Yaskawa INFORM job: A_ROOF_SIDE_0617_2_PAINT_61.JBI

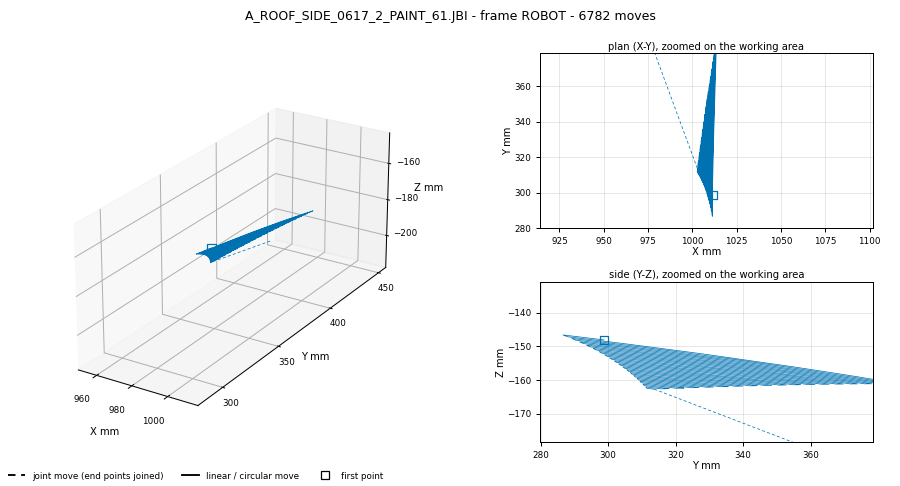
[picture p0: tool path of A_ROOF_SIDE_0617_2_PAINT_61.JBI in frame ROBOT, 6782 of 6782 moves have a stored position in this frame; points joined in program order, loops and branches not executed]
/JOB
//NAME A_ROOF_SIDE_0617_2_PAINT61
//POS
///NPOS 6782,0,0,0,0,0
///TOOL 1
///USER 0
///POSTYPE ROBOT
///RECTAN
///RCONF 1,0,0,0,0,0,0,0,0,0,0,0,0,0,0,0,0,0,0,0,0,0,0,0
C00000=1011.484,298.812,-148.095,169.236,53.491,160.314
C00001=1011.478,298.564,-148.065,169.230,53.497,160.314
C00002=1011.473,298.316,-148.034,169.223,53.504,160.314
C00003=1011.467,298.068,-148.004,169.218,53.510,160.315
C00004=1011.462,297.820,-147.973,169.211,53.517,160.315
C00005=1011.456,297.573,-147.942,169.204,53.524,160.315
C00006=1011.451,297.324,-147.911,169.198,53.530,160.315
C00007=1011.445,297.077,-147.881,169.192,53.537,160.315
C00008=1011.440,296.828,-147.850,169.186,53.544,160.316
C00009=1011.434,296.581,-147.820,169.180,53.551,160.316
C00010=1011.429,296.332,-147.789,169.174,53.558,160.316
C00011=1011.424,296.084,-147.759,169.167,53.565,160.316
C00012=1011.418,295.836,-147.728,169.161,53.572,160.317
C00013=1011.413,295.588,-147.698,169.155,53.578,160.317
C00014=1011.408,295.340,-147.667,169.148,53.585,160.317
C00015=1011.402,295.093,-147.637,169.142,53.592,160.317
C00016=1011.398,294.844,-147.607,169.136,53.599,160.317
C00017=1011.392,294.596,-147.576,169.130,53.605,160.318
C00018=1011.387,294.348,-147.545,169.123,53.612,160.318
C00019=1011.381,294.100,-147.515,169.117,53.620,160.318
C00020=1011.376,293.852,-147.485,169.111,53.626,160.319
C00021=1011.369,293.566,-147.450,169.104,53.634,160.319
C00022=1011.364,293.280,-147.415,169.097,53.642,160.319
C00023=1011.358,292.995,-147.380,169.090,53.650,160.319
C00024=1011.352,292.709,-147.345,169.082,53.658,160.320
C00025=1011.347,292.461,-147.315,169.077,53.665,160.320
C00026=1011.341,292.212,-147.285,169.070,53.672,160.320
C00027=1011.336,291.964,-147.255,169.065,53.679,160.321
C00028=1011.331,291.716,-147.225,169.058,53.686,160.321
C00029=1011.326,291.468,-147.194,169.051,53.693,160.321
C00030=1011.320,291.220,-147.165,169.046,53.700,160.321
C00031=1011.315,290.971,-147.135,169.039,53.707,160.322
C00032=1011.309,290.724,-147.105,169.034,53.714,160.322
C00033=1011.304,290.476,-147.075,169.027,53.721,160.322
C00034=1011.298,290.227,-147.046,169.021,53.728,160.322
C00035=1011.293,289.979,-147.015,169.015,53.736,160.323
C00036=1011.288,289.732,-146.986,169.009,53.742,160.323
C00037=1011.283,289.483,-146.956,169.002,53.750,160.324
C00038=1011.277,289.235,-146.926,168.997,53.757,160.324
C00039=1011.272,288.987,-146.897,168.990,53.764,160.324
C00040=1011.267,288.739,-146.867,168.985,53.771,160.324
C00041=1011.261,288.491,-146.837,168.979,53.779,160.325
C00042=1011.256,288.243,-146.808,168.972,53.785,160.325
C00043=1011.251,287.995,-146.778,168.967,53.793,160.325
C00044=1011.245,287.746,-146.749,168.960,53.800,160.326
C00045=1011.240,287.463,-146.715,168.953,53.808,160.326
C00046=1011.233,287.181,-146.682,168.946,53.816,160.326
C00047=1011.227,286.898,-146.648,168.940,53.824,160.327
C00048=1011.221,286.616,-146.614,168.933,53.833,160.327
C00049=1010.990,287.953,-147.138,168.938,53.865,160.336
C00050=1010.994,288.177,-147.165,168.944,53.858,160.335
C00051=1010.999,288.403,-147.191,168.949,53.852,160.335
C00052=1011.004,288.627,-147.218,168.955,53.845,160.335
C00053=1011.008,288.853,-147.245,168.961,53.839,160.335
C00054=1011.014,289.077,-147.272,168.965,53.832,160.334
C00055=1011.018,289.303,-147.299,168.971,53.826,160.334
C00056=1011.023,289.527,-147.326,168.977,53.819,160.334
C00057=1011.027,289.753,-147.353,168.983,53.813,160.334
C00058=1011.033,290.001,-147.382,168.989,53.806,160.333
C00059=1011.038,290.249,-147.412,168.995,53.799,160.333
C00060=1011.043,290.497,-147.442,169.001,53.792,160.333
C00061=1011.049,290.745,-147.471,169.007,53.785,160.332
C00062=1011.054,290.993,-147.501,169.013,53.778,160.332
C00063=1011.060,291.242,-147.531,169.020,53.770,160.332
C00064=1011.064,291.489,-147.561,169.025,53.764,160.332
C00065=1011.070,291.738,-147.591,169.032,53.756,160.331
C00066=1011.075,291.986,-147.621,169.038,53.749,160.331
C00067=1011.081,292.233,-147.651,169.044,53.743,160.331
C00068=1011.085,292.482,-147.681,169.051,53.736,160.331
C00069=1011.091,292.730,-147.711,169.056,53.728,160.330
C00070=1011.096,293.018,-147.746,169.063,53.720,160.330
C00071=1011.103,293.306,-147.781,169.070,53.712,160.330
C00072=1011.110,293.594,-147.817,169.078,53.704,160.329
C00073=1011.115,293.882,-147.852,169.085,53.696,160.329
C00074=1011.121,294.130,-147.882,169.092,53.689,160.329
C00075=1011.126,294.379,-147.913,169.097,53.683,160.329
C00076=1011.131,294.627,-147.943,169.104,53.676,160.328
C00077=1011.136,294.874,-147.973,169.111,53.669,160.328
C00078=1011.141,295.122,-148.003,169.117,53.662,160.328
C00079=1011.147,295.371,-148.034,169.123,53.655,160.328
C00080=1011.152,295.618,-148.064,169.128,53.648,160.327
C00081=1011.157,295.867,-148.095,169.135,53.641,160.327
C00082=1011.163,296.115,-148.125,169.141,53.635,160.327
C00083=1011.168,296.363,-148.156,169.148,53.628,160.327
C00084=1011.174,296.611,-148.186,169.154,53.621,160.327
C00085=1011.179,296.859,-148.217,169.160,53.614,160.326
C00086=1011.185,297.107,-148.248,169.167,53.607,160.326
C00087=1011.189,297.354,-148.278,169.172,53.601,160.326
C00088=1011.195,297.603,-148.308,169.179,53.594,160.326
C00089=1011.200,297.851,-148.339,169.186,53.587,160.326
C00090=1011.205,298.099,-148.370,169.192,53.581,160.325
C00091=1011.211,298.347,-148.400,169.198,53.574,160.325
C00092=1011.216,298.595,-148.431,169.204,53.567,160.325
C00093=1011.222,298.843,-148.461,169.211,53.560,160.325
C00094=1011.227,299.091,-148.492,169.218,53.554,160.325
C00095=1011.233,299.339,-148.523,169.224,53.547,160.324
C00096=1011.238,299.588,-148.554,169.230,53.540,160.324
C00097=1011.244,299.835,-148.584,169.237,53.534,160.324
C00098=1011.249,300.084,-148.615,169.243,53.527,160.324
C00099=1011.255,300.331,-148.646,169.250,53.520,160.324
C00100=1011.260,300.580,-148.676,169.255,53.514,160.323
C00101=1011.266,300.827,-148.707,169.262,53.507,160.323
C00102=1011.271,301.075,-148.738,169.269,53.500,160.323
C00103=1011.277,301.323,-148.769,169.275,53.494,160.323
C00104=1011.282,301.571,-148.800,169.282,53.487,160.323
C00105=1011.288,301.819,-148.831,169.287,53.480,160.323
C00106=1011.294,302.067,-148.861,169.295,53.474,160.323
C00107=1011.299,302.315,-148.892,169.301,53.467,160.322
C00108=1011.304,302.563,-148.923,169.307,53.461,160.322
C00109=1011.311,302.811,-148.954,169.314,53.454,160.322
C00110=1011.316,303.059,-148.985,169.321,53.448,160.322
C00111=1011.322,303.307,-149.015,169.327,53.441,160.322
C00112=1011.327,303.555,-149.046,169.333,53.434,160.322
C00113=1011.333,303.803,-149.077,169.340,53.428,160.322
C00114=1011.338,304.051,-149.108,169.346,53.422,160.321
C00115=1011.345,304.299,-149.139,169.353,53.415,160.321
C00116=1011.350,304.547,-149.171,169.359,53.409,160.321
C00117=1011.356,304.795,-149.201,169.366,53.402,160.321
C00118=1011.362,305.043,-149.233,169.373,53.395,160.321
C00119=1011.368,305.291,-149.264,169.379,53.389,160.321
C00120=1011.373,305.539,-149.294,169.386,53.382,160.321
C00121=1011.380,305.787,-149.326,169.393,53.376,160.321
C00122=1011.385,306.035,-149.357,169.398,53.370,160.320
C00123=1011.391,306.282,-149.388,169.405,53.363,160.320
C00124=1011.396,306.531,-149.419,169.412,53.356,160.320
C00125=1011.403,306.778,-149.450,169.418,53.350,160.320
C00126=1011.408,307.026,-149.481,169.425,53.344,160.320
C00127=1011.414,307.274,-149.513,169.432,53.337,160.320
C00128=1011.419,307.522,-149.544,169.438,53.331,160.320
C00129=1011.425,307.770,-149.576,169.445,53.325,160.320
C00130=1011.433,308.076,-149.614,169.454,53.316,160.320
C00131=1011.440,308.383,-149.652,169.461,53.309,160.320
C00132=1011.448,308.689,-149.691,169.470,53.301,160.319
C00133=1011.455,308.995,-149.730,169.479,53.293,160.319
C00134=1011.460,309.243,-149.762,169.484,53.287,160.319
C00135=1011.465,309.491,-149.794,169.491,53.281,160.319
C00136=1011.471,309.739,-149.826,169.498,53.275,160.319
C00137=1011.476,309.986,-149.858,169.505,53.269,160.319
C00138=1011.482,310.235,-149.890,169.511,53.263,160.319
C00139=1011.488,310.481,-149.922,169.518,53.256,160.319
C00140=1011.494,310.730,-149.954,169.525,53.250,160.319
C00141=1011.498,310.977,-149.986,169.531,53.244,160.319
C00142=1011.504,311.226,-150.019,169.538,53.238,160.319
C00143=1011.510,311.473,-150.050,169.545,53.232,160.319
C00144=1011.516,311.721,-150.082,169.551,53.225,160.319
C00145=1011.521,311.969,-150.114,169.559,53.219,160.319
C00146=1011.528,312.216,-150.147,169.565,53.213,160.319
C00147=1011.533,312.464,-150.178,169.572,53.207,160.319
C00148=1011.538,312.713,-150.211,169.578,53.201,160.319
C00149=1011.544,312.961,-150.243,169.585,53.195,160.319
C00150=1011.550,313.208,-150.275,169.592,53.189,160.319
C00151=1011.556,313.456,-150.307,169.599,53.183,160.319
C00152=1011.561,313.703,-150.339,169.606,53.177,160.319
C00153=1011.567,313.951,-150.372,169.612,53.171,160.319
C00154=1011.573,314.199,-150.404,169.619,53.165,160.319
C00155=1011.578,314.447,-150.436,169.627,53.158,160.319
C00156=1011.584,314.695,-150.469,169.633,53.153,160.319
C00157=1011.590,314.943,-150.501,169.640,53.146,160.319
C00158=1011.597,315.190,-150.534,169.646,53.141,160.319
C00159=1011.601,315.438,-150.566,169.653,53.134,160.319
C00160=1011.608,315.686,-150.599,169.661,53.128,160.319
C00161=1011.614,315.934,-150.631,169.667,53.123,160.319
C00162=1011.620,316.182,-150.663,169.674,53.116,160.319
C00163=1011.625,316.429,-150.695,169.681,53.110,160.319
C00164=1011.632,316.677,-150.728,169.688,53.105,160.319
C00165=1011.637,316.925,-150.760,169.695,53.099,160.319
C00166=1011.643,317.173,-150.793,169.701,53.093,160.319
C00167=1011.649,317.421,-150.825,169.709,53.087,160.319
C00168=1011.655,317.668,-150.857,169.716,53.081,160.319
C00169=1011.661,317.916,-150.890,169.722,53.076,160.319
C00170=1011.667,318.164,-150.922,169.730,53.069,160.319
C00171=1011.673,318.412,-150.956,169.737,53.063,160.319
C00172=1011.679,318.659,-150.988,169.743,53.057,160.319
C00173=1011.685,318.907,-151.020,169.751,53.052,160.319
C00174=1011.691,319.155,-151.053,169.758,53.046,160.320
C00175=1011.698,319.403,-151.086,169.764,53.040,160.319
C00176=1011.703,319.651,-151.118,169.771,53.034,160.319
C00177=1011.709,319.899,-151.151,169.779,53.028,160.320
C00178=1011.715,320.146,-151.184,169.785,53.023,160.320
C00179=1011.722,320.394,-151.217,169.792,53.016,160.320
C00180=1011.728,320.642,-151.249,169.800,53.011,160.320
C00181=1011.734,320.889,-151.282,169.806,53.005,160.320
C00182=1011.739,321.138,-151.315,169.814,53.000,160.320
C00183=1011.746,321.385,-151.348,169.821,52.994,160.320
C00184=1011.752,321.633,-151.380,169.827,52.988,160.320
C00185=1011.758,321.880,-151.413,169.835,52.982,160.320
C00186=1011.765,322.128,-151.446,169.842,52.976,160.320
C00187=1011.770,322.376,-151.479,169.849,52.971,160.321
C00188=1011.777,322.624,-151.512,169.856,52.965,160.321
C00189=1011.783,322.871,-151.545,169.864,52.959,160.321
C00190=1011.791,323.183,-151.586,169.873,52.952,160.321
C00191=1011.799,323.495,-151.627,169.882,52.945,160.321
C00192=1011.807,323.807,-151.669,169.891,52.938,160.321
C00193=1011.815,324.119,-151.711,169.900,52.931,160.322
C00194=1011.821,324.366,-151.743,169.906,52.925,160.321
C00195=1011.827,324.614,-151.776,169.914,52.920,160.322
C00196=1011.833,324.862,-151.810,169.921,52.914,160.322
C00197=1011.839,325.109,-151.842,169.929,52.908,160.322
C00198=1011.847,325.357,-151.876,169.936,52.903,160.322
C00199=1011.853,325.604,-151.909,169.943,52.897,160.322
C00200=1011.859,325.852,-151.943,169.951,52.891,160.322
C00201=1011.864,326.100,-151.976,169.957,52.886,160.323
C00202=1011.871,326.347,-152.010,169.965,52.881,160.323
C00203=1011.877,326.595,-152.043,169.973,52.875,160.323
C00204=1011.883,326.843,-152.077,169.979,52.870,160.323
C00205=1011.889,327.090,-152.110,169.986,52.864,160.323
C00206=1011.896,327.338,-152.145,169.994,52.859,160.324
C00207=1011.901,327.586,-152.178,170.001,52.854,160.324
C00208=1011.908,327.833,-152.211,170.008,52.848,160.324
C00209=1011.914,328.081,-152.246,170.016,52.843,160.324
C00210=1011.920,328.329,-152.279,170.023,52.838,160.324
C00211=1011.926,328.576,-152.313,170.030,52.832,160.325
C00212=1011.933,328.824,-152.347,170.038,52.827,160.325
C00213=1011.939,329.071,-152.380,170.046,52.821,160.325
C00214=1011.946,329.319,-152.414,170.052,52.816,160.325
C00215=1011.951,329.567,-152.448,170.060,52.811,160.325
C00216=1011.958,329.814,-152.481,170.068,52.805,160.326
C00217=1011.964,330.062,-152.515,170.074,52.800,160.326
C00218=1011.970,330.310,-152.550,170.082,52.795,160.326
C00219=1011.977,330.557,-152.583,170.090,52.789,160.326
C00220=1011.983,330.804,-152.617,170.097,52.784,160.327
C00221=1011.990,331.052,-152.652,170.104,52.778,160.327
C00222=1011.996,331.299,-152.685,170.112,52.773,160.327
C00223=1012.002,331.548,-152.719,170.119,52.768,160.327
C00224=1012.008,331.795,-152.753,170.127,52.762,160.327
C00225=1012.016,332.042,-152.788,170.134,52.757,160.328
C00226=1012.022,332.290,-152.822,170.142,52.752,160.328
C00227=1012.028,332.538,-152.856,170.150,52.747,160.328
C00228=1012.034,332.786,-152.890,170.156,52.742,160.328
C00229=1012.040,333.033,-152.924,170.164,52.736,160.329
C00230=1012.047,333.281,-152.959,170.172,52.731,160.329
C00231=1012.053,333.528,-152.993,170.180,52.726,160.329
C00232=1012.059,333.776,-153.028,170.186,52.721,160.330
C00233=1012.066,334.024,-153.063,170.194,52.716,160.330
C00234=1012.072,334.271,-153.097,170.202,52.711,160.330
C00235=1012.079,334.519,-153.130,170.210,52.705,160.330
C00236=1012.086,334.766,-153.166,170.217,52.701,160.331
C00237=1012.092,335.013,-153.200,170.225,52.695,160.331
C00238=1012.098,335.261,-153.234,170.233,52.691,160.332
C00239=1012.105,335.509,-153.269,170.240,52.685,160.332
C00240=1012.111,335.756,-153.303,170.248,52.681,160.332
C00241=1012.117,336.003,-153.338,170.255,52.675,160.332
C00242=1012.124,336.251,-153.373,170.263,52.670,160.333
C00243=1012.130,336.499,-153.407,170.271,52.665,160.333
C00244=1012.137,336.746,-153.442,170.278,52.661,160.333
C00245=1012.144,336.993,-153.476,170.286,52.655,160.334
C00246=1012.150,337.241,-153.511,170.294,52.650,160.334
C00247=1012.157,337.489,-153.545,170.302,52.645,160.334
C00248=1012.164,337.736,-153.580,170.310,52.640,160.335
C00249=1012.170,337.984,-153.616,170.316,52.635,160.335
C00250=1012.178,338.291,-153.658,170.326,52.629,160.335
C00251=1012.186,338.599,-153.702,170.336,52.623,160.336
C00252=1012.194,338.907,-153.745,170.346,52.617,160.337
C00253=1012.202,339.213,-153.789,170.355,52.611,160.337
C00254=1012.209,339.461,-153.824,170.364,52.606,160.337
C00255=1012.216,339.708,-153.859,170.371,52.601,160.338
C00256=1012.223,339.956,-153.894,170.378,52.596,160.338
C00257=1012.229,340.203,-153.930,170.386,52.591,160.338
C00258=1012.235,340.451,-153.965,170.395,52.587,160.339
C00259=1012.242,340.699,-154.000,170.403,52.582,160.339
C00260=1012.249,340.946,-154.035,170.410,52.576,160.340
C00261=1012.255,341.193,-154.070,170.418,52.572,160.340
C00262=1012.262,341.441,-154.105,170.426,52.567,160.340
C00263=1012.268,341.688,-154.141,170.434,52.562,160.341
C00264=1012.275,341.935,-154.177,170.442,52.558,160.341
C00265=1012.282,342.182,-154.212,170.450,52.553,160.342
C00266=1012.289,342.430,-154.247,170.458,52.548,160.342
C00267=1012.296,342.677,-154.282,170.465,52.544,160.343
C00268=1012.302,342.925,-154.318,170.473,52.539,160.343
C00269=1012.309,343.173,-154.353,170.481,52.534,160.344
C00270=1012.316,343.420,-154.389,170.490,52.529,160.344
C00271=1012.323,343.667,-154.424,170.498,52.525,160.344
C00272=1012.329,343.915,-154.460,170.506,52.520,160.345
C00273=1012.336,344.162,-154.495,170.514,52.515,160.345
C00274=1012.343,344.409,-154.531,170.521,52.511,160.346
C00275=1012.350,344.657,-154.566,170.530,52.506,160.346
C00276=1012.356,344.905,-154.602,170.538,52.502,160.347
C00277=1012.363,345.151,-154.638,170.546,52.497,160.347
C00278=1012.370,345.399,-154.673,170.554,52.492,160.348
C00279=1012.378,345.646,-154.709,170.562,52.487,160.348
C00280=1012.384,345.894,-154.745,170.571,52.483,160.349
C00281=1012.391,346.141,-154.781,170.579,52.478,160.349
C00282=1012.397,346.388,-154.816,170.587,52.474,160.350
C00283=1012.404,346.636,-154.853,170.594,52.469,160.350
C00284=1012.411,346.883,-154.888,170.602,52.465,160.351
C00285=1012.417,347.130,-154.924,170.611,52.460,160.351
C00286=1012.425,347.378,-154.961,170.619,52.456,160.352
C00287=1012.431,347.625,-154.996,170.627,52.451,160.352
C00288=1012.438,347.872,-155.032,170.635,52.447,160.353
C00289=1012.445,348.120,-155.069,170.644,52.443,160.353
C00290=1012.452,348.366,-155.105,170.652,52.438,160.354
C00291=1012.459,348.614,-155.142,170.661,52.434,160.355
C00292=1012.466,348.862,-155.177,170.669,52.429,160.355
C00293=1012.472,349.109,-155.213,170.676,52.425,160.356
C00294=1012.480,349.356,-155.250,170.684,52.420,160.356
C00295=1012.486,349.603,-155.286,170.693,52.416,160.357
C00296=1012.494,349.851,-155.322,170.701,52.412,160.357
C00297=1012.500,350.098,-155.359,170.710,52.407,160.358
C00298=1012.508,350.345,-155.395,170.718,52.403,160.358
C00299=1012.514,350.592,-155.431,170.726,52.399,160.359
C00300=1012.522,350.840,-155.468,170.735,52.394,160.360
C00301=1012.528,351.087,-155.504,170.743,52.390,160.360
C00302=1012.536,351.334,-155.540,170.751,52.386,160.361
C00303=1012.543,351.582,-155.577,170.760,52.381,160.361
C00304=1012.550,351.828,-155.614,170.768,52.377,160.362
C00305=1012.557,352.076,-155.650,170.777,52.373,160.362
C00306=1012.564,352.322,-155.686,170.785,52.368,160.363
C00307=1012.571,352.570,-155.723,170.794,52.364,160.364
C00308=1012.579,352.818,-155.759,170.802,52.360,160.364
C00309=1012.586,353.064,-155.796,170.810,52.355,160.365
C00310=1012.594,353.369,-155.842,170.821,52.351,160.366
C00311=1012.603,353.675,-155.887,170.832,52.346,160.367
C00312=1012.612,353.979,-155.932,170.842,52.340,160.367
C00313=1012.621,354.284,-155.978,170.852,52.335,160.368
C00314=1012.628,354.531,-156.015,170.861,52.331,160.369
C00315=1012.634,354.778,-156.052,170.869,52.327,160.369
C00316=1012.642,355.025,-156.089,170.879,52.322,160.370
C00317=1012.649,355.273,-156.125,170.887,52.318,160.371
C00318=1012.657,355.520,-156.163,170.896,52.314,160.371
C00319=1012.665,355.767,-156.200,170.904,52.310,160.372
C00320=1012.671,356.014,-156.236,170.913,52.306,160.373
C00321=1012.678,356.261,-156.274,170.922,52.302,160.373
C00322=1012.685,356.508,-156.311,170.930,52.298,160.374
C00323=1012.693,356.756,-156.348,170.939,52.294,160.375
C00324=1012.700,357.003,-156.385,170.948,52.290,160.376
C00325=1012.708,357.250,-156.423,170.956,52.286,160.376
C00326=1012.715,357.497,-156.460,170.965,52.282,160.377
C00327=1012.723,357.744,-156.497,170.973,52.278,160.378
C00328=1012.730,357.992,-156.534,170.982,52.274,160.378
C00329=1012.737,358.239,-156.571,170.991,52.270,160.379
C00330=1012.744,358.486,-156.609,171.000,52.266,160.380
C00331=1012.752,358.733,-156.647,171.009,52.262,160.381
C00332=1012.758,358.979,-156.684,171.018,52.258,160.381
C00333=1012.766,359.226,-156.722,171.026,52.254,160.382
C00334=1012.773,359.473,-156.759,171.035,52.251,160.383
C00335=1012.781,359.721,-156.797,171.044,52.247,160.384
C00336=1012.788,359.968,-156.835,171.053,52.243,160.384
C00337=1012.795,360.215,-156.872,171.061,52.239,160.385
C00338=1012.803,360.462,-156.911,171.070,52.235,160.386
C00339=1012.810,360.709,-156.948,171.080,52.231,160.387
C00340=1012.817,360.956,-156.986,171.089,52.227,160.388
C00341=1012.825,361.203,-157.024,171.098,52.224,160.389
C00342=1012.832,361.450,-157.061,171.106,52.220,160.389
C00343=1012.839,361.697,-157.099,171.115,52.216,160.390
C00344=1012.847,361.943,-157.137,171.124,52.212,160.391
C00345=1012.855,362.191,-157.175,171.134,52.208,160.392
C00346=1012.862,362.438,-157.213,171.143,52.205,160.393
C00347=1012.870,362.685,-157.251,171.151,52.201,160.393
C00348=1012.877,362.931,-157.289,171.160,52.197,160.394
C00349=1012.885,363.179,-157.327,171.169,52.194,160.395
C00350=1012.892,363.426,-157.365,171.179,52.190,160.396
C00351=1012.900,363.673,-157.403,171.188,52.186,160.397
C00352=1012.907,363.919,-157.441,171.197,52.183,160.397
C00353=1012.915,364.167,-157.480,171.206,52.179,160.398
C00354=1012.923,364.414,-157.517,171.216,52.175,160.399
C00355=1012.930,364.660,-157.555,171.225,52.172,160.400
C00356=1012.938,364.907,-157.594,171.234,52.168,160.401
C00357=1012.946,365.155,-157.632,171.243,52.165,160.402
C00358=1012.954,365.402,-157.670,171.253,52.161,160.403
C00359=1012.961,365.648,-157.708,171.262,52.157,160.404
C00360=1012.969,365.895,-157.747,171.271,52.154,160.405
C00361=1012.977,366.142,-157.785,171.280,52.151,160.405
C00362=1012.985,366.389,-157.824,171.290,52.147,160.406
C00363=1012.993,366.636,-157.862,171.299,52.143,160.407
C00364=1013.000,366.883,-157.901,171.308,52.140,160.408
C00365=1013.008,367.130,-157.940,171.318,52.136,160.409
C00366=1013.015,367.376,-157.978,171.327,52.132,160.410
C00367=1013.023,367.624,-158.017,171.336,52.129,160.411
C00368=1013.030,367.870,-158.055,171.346,52.126,160.412
C00369=1013.039,368.117,-158.095,171.355,52.122,160.413
C00370=1013.048,368.429,-158.144,171.367,52.118,160.414
C00371=1013.057,368.742,-158.193,171.379,52.114,160.415
C00372=1013.067,369.055,-158.242,171.390,52.109,160.416
C00373=1013.077,369.367,-158.291,171.403,52.105,160.418
C00374=1013.085,369.614,-158.331,171.413,52.102,160.419
C00375=1013.093,369.860,-158.369,171.422,52.098,160.420
C00376=1013.101,370.107,-158.409,171.431,52.095,160.421
C00377=1013.108,370.355,-158.448,171.441,52.091,160.422
C00378=1013.117,370.601,-158.487,171.450,52.089,160.423
C00379=1013.124,370.848,-158.525,171.460,52.085,160.424
C00380=1013.132,371.095,-158.565,171.470,52.082,160.425
C00381=1013.140,371.342,-158.604,171.479,52.078,160.426
C00382=1013.149,371.588,-158.643,171.489,52.075,160.427
C00383=1013.156,371.835,-158.683,171.498,52.072,160.428
C00384=1013.164,372.082,-158.721,171.508,52.068,160.429
C00385=1013.172,372.329,-158.761,171.518,52.066,160.430
C00386=1013.180,372.575,-158.801,171.528,52.062,160.431
C00387=1013.189,372.822,-158.840,171.537,52.059,160.432
C00388=1013.196,373.069,-158.879,171.548,52.056,160.433
C00389=1013.205,373.316,-158.918,171.557,52.053,160.434
C00390=1013.212,373.562,-158.957,171.567,52.049,160.435
C00391=1013.220,373.809,-158.997,171.576,52.046,160.436
C00392=1013.229,374.055,-159.037,171.587,52.043,160.438
C00393=1013.237,374.302,-159.076,171.596,52.040,160.439
C00394=1013.245,374.549,-159.116,171.606,52.037,160.440
C00395=1013.253,374.796,-159.155,171.616,52.034,160.441
C00396=1013.262,375.042,-159.195,171.626,52.031,160.442
C00397=1013.269,375.289,-159.234,171.636,52.028,160.443
C00398=1013.277,375.536,-159.274,171.646,52.025,160.444
C00399=1013.285,375.782,-159.315,171.655,52.022,160.445
C00400=1013.294,376.030,-159.355,171.666,52.019,160.447
C00401=1013.302,376.276,-159.395,171.676,52.015,160.448
C00402=1013.310,376.523,-159.435,171.686,52.013,160.449
C00403=1013.318,376.769,-159.475,171.696,52.009,160.450
C00404=1013.326,377.016,-159.515,171.705,52.007,160.451
C00405=1013.334,377.263,-159.555,171.716,52.004,160.453
C00406=1013.343,377.508,-159.595,171.727,52.001,160.454
C00407=1013.351,377.755,-159.635,171.736,51.998,160.455
C00408=1013.359,378.002,-159.676,171.746,51.995,160.456
C00409=1013.368,378.249,-159.715,171.756,51.992,160.457
C00410=1013.376,378.495,-159.756,171.767,51.989,160.458
C00411=1013.384,378.742,-159.797,171.777,51.986,160.460
C00412=1013.392,378.988,-159.837,171.787,51.984,160.461
C00413=1013.401,379.235,-159.877,171.797,51.980,160.462
C00414=1013.409,379.481,-159.918,171.808,51.978,160.463
C00415=1013.417,379.728,-159.958,171.817,51.975,160.465
C00416=1013.426,379.975,-159.998,171.828,51.972,160.466
C00417=1013.434,380.221,-160.039,171.839,51.969,160.467
C00418=1013.442,380.468,-160.079,171.849,51.967,160.468
C00419=1013.451,380.714,-160.120,171.859,51.964,160.470
C00420=1013.459,380.961,-160.160,171.870,51.961,160.471
C00421=1013.468,381.207,-160.201,171.880,51.958,160.472
C00422=1013.477,381.453,-160.241,171.891,51.955,160.473
C00423=1013.485,381.700,-160.282,171.901,51.953,160.475
C00424=1013.493,381.947,-160.323,171.911,51.950,160.476
C00425=1013.503,382.193,-160.363,171.922,51.947,160.477
C00426=1013.511,382.440,-160.404,171.933,51.945,160.479
C00427=1013.520,382.687,-160.445,171.943,51.942,160.480
C00428=1013.528,382.933,-160.485,171.954,51.939,160.481
C00429=1013.537,383.179,-160.527,171.964,51.936,160.483
C00430=1013.548,383.480,-160.577,171.977,51.934,160.484
C00431=1013.558,383.781,-160.627,171.990,51.930,160.486
C00432=1013.569,384.083,-160.677,172.003,51.927,160.488
C00433=1013.580,384.384,-160.727,172.017,51.924,160.489
C00434=1013.588,384.631,-160.768,172.027,51.921,160.491
C00435=1013.597,384.877,-160.809,172.037,51.919,160.492
C00436=1013.606,385.124,-160.850,172.048,51.916,160.494
C00437=1013.615,385.370,-160.892,172.059,51.914,160.495
C00438=1013.623,385.616,-160.933,172.070,51.911,160.496
C00439=1013.632,385.863,-160.974,172.080,51.908,160.498
C00440=1013.640,386.109,-161.016,172.092,51.906,160.499
C00441=1013.649,386.356,-161.058,172.103,51.904,160.501
C00442=1013.305,384.294,-161.060,171.994,51.982,160.501
C00443=1013.295,384.035,-161.017,171.984,51.985,160.499
C00444=1013.286,383.776,-160.974,171.972,51.988,160.498
C00445=1013.277,383.517,-160.931,171.961,51.991,160.496
C00446=1013.268,383.257,-160.887,171.949,51.994,160.495
C00447=1013.259,383.011,-160.847,171.939,51.996,160.494
C00448=1013.250,382.764,-160.806,171.929,51.999,160.492
C00449=1013.242,382.518,-160.765,171.918,52.001,160.491
C00450=1013.233,382.271,-160.725,171.907,52.005,160.490
C00451=1013.225,382.025,-160.684,171.897,52.007,160.488
C00452=1013.216,381.778,-160.643,171.886,52.010,160.487
C00453=1013.208,381.532,-160.603,171.875,52.013,160.486
C00454=1013.200,381.285,-160.563,171.865,52.015,160.484
C00455=1013.191,381.038,-160.522,171.855,52.018,160.483
C00456=1013.182,380.792,-160.482,171.844,52.021,160.482
C00457=1013.174,380.545,-160.441,171.833,52.024,160.480
C00458=1013.165,380.299,-160.400,171.824,52.027,160.479
C00459=1013.157,380.053,-160.360,171.813,52.029,160.478
C00460=1013.148,379.806,-160.320,171.803,52.032,160.477
C00461=1013.140,379.559,-160.279,171.792,52.035,160.475
C00462=1013.132,379.313,-160.239,171.783,52.038,160.474
C00463=1013.123,379.066,-160.198,171.772,52.041,160.473
C00464=1013.115,378.819,-160.158,171.761,52.044,160.472
C00465=1013.107,378.573,-160.118,171.751,52.047,160.470
C00466=1013.099,378.326,-160.078,171.742,52.050,160.469
C00467=1013.090,378.079,-160.037,171.731,52.052,160.468
C00468=1013.082,377.833,-159.998,171.721,52.056,160.467
C00469=1013.074,377.587,-159.957,171.711,52.059,160.466
C00470=1013.066,377.340,-159.917,171.701,52.062,160.465
C00471=1013.058,377.093,-159.876,171.690,52.064,160.463
C00472=1013.049,376.847,-159.837,171.680,52.067,160.462
C00473=1013.041,376.601,-159.797,171.670,52.071,160.461
C00474=1013.034,376.354,-159.757,171.661,52.073,160.460
C00475=1013.025,376.107,-159.717,171.650,52.077,160.459
C00476=1013.017,375.861,-159.677,171.640,52.080,160.457
C00477=1013.009,375.613,-159.636,171.631,52.083,160.456
C00478=1013.001,375.367,-159.597,171.620,52.086,160.455
C00479=1012.993,375.120,-159.557,171.611,52.089,160.454
C00480=1012.985,374.874,-159.517,171.600,52.092,160.453
C00481=1012.977,374.627,-159.478,171.591,52.095,160.452
C00482=1012.969,374.380,-159.439,171.581,52.098,160.451
C00483=1012.961,374.133,-159.399,171.570,52.101,160.449
C00484=1012.953,373.887,-159.360,171.561,52.104,160.448
C00485=1012.944,373.640,-159.320,171.551,52.108,160.447
C00486=1012.936,373.393,-159.280,171.541,52.111,160.446
C00487=1012.928,373.147,-159.241,171.531,52.114,160.445
C00488=1012.919,372.900,-159.202,171.522,52.117,160.444
C00489=1012.912,372.653,-159.163,171.512,52.121,160.443
C00490=1012.904,372.406,-159.123,171.502,52.124,160.442
C00491=1012.895,372.159,-159.084,171.492,52.128,160.441
C00492=1012.888,371.913,-159.045,171.483,52.130,160.440
C00493=1012.880,371.666,-159.006,171.473,52.134,160.439
C00494=1012.872,371.419,-158.966,171.464,52.137,160.438
C00495=1012.864,371.172,-158.927,171.453,52.140,160.437
C00496=1012.856,370.926,-158.888,171.444,52.144,160.436
C00497=1012.849,370.678,-158.849,171.434,52.147,160.435
C00498=1012.840,370.432,-158.810,171.425,52.151,160.434
C00499=1012.833,370.185,-158.772,171.414,52.154,160.433
C00500=1012.825,369.938,-158.732,171.405,52.157,160.432
C00501=1012.817,369.691,-158.693,171.396,52.160,160.431
C00502=1012.809,369.445,-158.654,171.386,52.164,160.430
C00503=1012.799,369.130,-158.604,171.374,52.169,160.429
C00504=1012.789,368.815,-158.555,171.362,52.173,160.427
C00505=1012.779,368.500,-158.505,171.350,52.177,160.426
C00506=1012.770,368.186,-158.455,171.338,52.182,160.425
C00507=1012.762,367.939,-158.417,171.328,52.185,160.424
C00508=1012.754,367.692,-158.378,171.319,52.188,160.423
C00509=1012.747,367.445,-158.339,171.309,52.192,160.422
C00510=1012.739,367.198,-158.301,171.300,52.196,160.421
C00511=1012.731,366.951,-158.263,171.292,52.199,160.420
C00512=1012.724,366.704,-158.223,171.281,52.202,160.419
C00513=1012.717,366.457,-158.185,171.272,52.206,160.418
C00514=1012.709,366.211,-158.147,171.263,52.209,160.417
C00515=1012.701,365.964,-158.108,171.253,52.213,160.416
C00516=1012.693,365.717,-158.070,171.244,52.217,160.415
C00517=1012.685,365.470,-158.031,171.236,52.221,160.415
C00518=1012.678,365.223,-157.994,171.226,52.225,160.414
C00519=1012.670,364.976,-157.955,171.217,52.228,160.413
C00520=1012.662,364.729,-157.917,171.208,52.232,160.412
C00521=1012.655,364.482,-157.880,171.198,52.235,160.411
C00522=1012.647,364.235,-157.841,171.189,52.239,160.410
C00523=1012.639,363.988,-157.803,171.180,52.242,160.409
C00524=1012.632,363.741,-157.765,171.171,52.246,160.408
C00525=1012.624,363.495,-157.727,171.161,52.250,160.408
C00526=1012.617,363.247,-157.689,171.152,52.254,160.407
C00527=1012.609,363.000,-157.651,171.143,52.257,160.406
C00528=1012.602,362.753,-157.613,171.134,52.261,160.405
C00529=1012.594,362.507,-157.575,171.125,52.265,160.404
C00530=1012.587,362.259,-157.537,171.116,52.269,160.403
C00531=1012.579,362.012,-157.499,171.107,52.272,160.402
C00532=1012.572,361.765,-157.461,171.098,52.276,160.402
C00533=1012.564,361.518,-157.424,171.088,52.280,160.401
C00534=1012.557,361.271,-157.386,171.080,52.284,160.400
C00535=1012.550,361.024,-157.348,171.071,52.288,160.399
C00536=1012.542,360.777,-157.311,171.062,52.292,160.399
C00537=1012.535,360.531,-157.272,171.053,52.295,160.398
C00538=1012.528,360.283,-157.235,171.045,52.300,160.397
C00539=1012.520,360.036,-157.197,171.035,52.303,160.396
C00540=1012.513,359.789,-157.160,171.026,52.308,160.395
C00541=1012.506,359.542,-157.122,171.017,52.311,160.395
C00542=1012.499,359.295,-157.085,171.009,52.315,160.394
C00543=1012.491,359.048,-157.046,171.000,52.319,160.393
C00544=1012.484,358.801,-157.009,170.991,52.323,160.392
C00545=1012.477,358.554,-156.971,170.982,52.327,160.392
C00546=1012.469,358.307,-156.934,170.973,52.331,160.391
C00547=1012.462,358.059,-156.897,170.964,52.335,160.390
C00548=1012.455,357.812,-156.859,170.956,52.339,160.389
C00549=1012.448,357.565,-156.822,170.947,52.343,160.389
C00550=1012.440,357.318,-156.785,170.938,52.347,160.388
C00551=1012.433,357.071,-156.747,170.930,52.351,160.387
C00552=1012.426,356.823,-156.711,170.921,52.355,160.387
C00553=1012.418,356.576,-156.673,170.911,52.359,160.386
C00554=1012.411,356.330,-156.637,170.903,52.363,160.385
C00555=1012.404,356.082,-156.600,170.894,52.368,160.384
C00556=1012.397,355.835,-156.562,170.886,52.372,160.384
C00557=1012.390,355.588,-156.525,170.877,52.376,160.383
C00558=1012.382,355.341,-156.489,170.869,52.380,160.382
C00559=1012.375,355.094,-156.451,170.860,52.384,160.382
C00560=1012.368,354.846,-156.415,170.852,52.388,160.381
C00561=1012.360,354.600,-156.378,170.843,52.392,160.380
C00562=1012.353,354.352,-156.341,170.835,52.396,160.380
C00563=1012.345,354.045,-156.295,170.823,52.402,160.379
C00564=1012.336,353.738,-156.249,170.812,52.407,160.378
C00565=1012.327,353.430,-156.204,170.802,52.412,160.377
C00566=1012.319,353.124,-156.158,170.792,52.417,160.376
C00567=1012.311,352.876,-156.122,170.783,52.421,160.376
C00568=1012.304,352.630,-156.084,170.775,52.425,160.375
C00569=1012.298,352.382,-156.048,170.767,52.430,160.375
C00570=1012.290,352.135,-156.011,170.758,52.434,160.374
C00571=1012.283,351.888,-155.975,170.749,52.438,160.373
C00572=1012.276,351.640,-155.939,170.741,52.443,160.373
C00573=1012.269,351.393,-155.902,170.733,52.447,160.372
C00574=1012.262,351.146,-155.866,170.724,52.451,160.372
C00575=1012.255,350.899,-155.830,170.716,52.456,160.371
C00576=1012.248,350.651,-155.793,170.708,52.460,160.370
C00577=1012.241,350.404,-155.757,170.699,52.464,160.370
C00578=1012.234,350.157,-155.721,170.691,52.469,160.369
C00579=1012.227,349.910,-155.684,170.682,52.473,160.369
C00580=1012.220,349.662,-155.648,170.674,52.478,160.368
C00581=1012.213,349.415,-155.612,170.666,52.482,160.368
C00582=1012.206,349.168,-155.575,170.658,52.487,160.367
C00583=1012.199,348.921,-155.539,170.649,52.491,160.366
C00584=1012.192,348.672,-155.503,170.641,52.496,160.366
C00585=1012.186,348.425,-155.467,170.632,52.500,160.365
C00586=1012.179,348.179,-155.431,170.624,52.505,160.365
C00587=1012.172,347.931,-155.394,170.616,52.509,160.364
C00588=1012.165,347.684,-155.359,170.608,52.514,160.364
C00589=1012.159,347.436,-155.323,170.599,52.518,160.363
C00590=1012.151,347.189,-155.287,170.591,52.523,160.363
C00591=1012.144,346.942,-155.251,170.583,52.527,160.362
C00592=1012.138,346.695,-155.215,170.574,52.532,160.361
C00593=1012.130,346.447,-155.179,170.566,52.536,160.361
C00594=1012.124,346.199,-155.143,170.558,52.541,160.361
C00595=1012.117,345.953,-155.107,170.551,52.546,160.360
C00596=1012.110,345.705,-155.072,170.542,52.550,160.360
C00597=1012.104,345.458,-155.036,170.534,52.554,160.359
C00598=1012.097,345.210,-155.000,170.526,52.559,160.359
C00599=1012.090,344.963,-154.965,170.518,52.564,160.358
C00600=1012.083,344.716,-154.929,170.510,52.569,160.358
C00601=1012.077,344.468,-154.893,170.502,52.574,160.357
C00602=1012.070,344.221,-154.858,170.493,52.578,160.357
C00603=1012.063,343.973,-154.823,170.485,52.583,160.356
C00604=1012.055,343.726,-154.787,170.477,52.587,160.356
C00605=1012.049,343.479,-154.751,170.469,52.592,160.355
C00606=1012.043,343.231,-154.716,170.462,52.597,160.355
C00607=1012.036,342.984,-154.681,170.454,52.601,160.354
C00608=1012.029,342.737,-154.646,170.446,52.606,160.354
C00609=1012.023,342.489,-154.610,170.438,52.611,160.353
C00610=1012.016,342.242,-154.574,170.429,52.616,160.353
C00611=1012.009,341.995,-154.539,170.421,52.620,160.353
C00612=1012.003,341.747,-154.504,170.413,52.625,160.352
C00613=1011.996,341.500,-154.469,170.407,52.630,160.352
C00614=1011.990,341.252,-154.433,170.398,52.635,160.352
C00615=1011.983,341.005,-154.398,170.390,52.640,160.351
C00616=1011.976,340.758,-154.363,170.382,52.645,160.351
C00617=1011.970,340.510,-154.328,170.374,52.650,160.350
C00618=1011.963,340.262,-154.293,170.366,52.654,160.350
C00619=1011.956,340.015,-154.258,170.358,52.660,160.349
C00620=1011.950,339.767,-154.222,170.351,52.664,160.349
C00621=1011.943,339.520,-154.187,170.343,52.669,160.349
C00622=1011.937,339.272,-154.152,170.335,52.674,160.348
C00623=1011.929,338.963,-154.109,170.325,52.680,160.348
C00624=1011.920,338.653,-154.064,170.316,52.686,160.347
C00625=1011.912,338.343,-154.021,170.306,52.692,160.347
C00626=1011.904,338.033,-153.978,170.296,52.699,160.346
C00627=1011.898,337.786,-153.943,170.288,52.703,160.346
C00628=1011.891,337.538,-153.908,170.280,52.709,160.346
C00629=1011.884,337.291,-153.873,170.272,52.714,160.345
C00630=1011.878,337.043,-153.839,170.266,52.719,160.345
C00631=1011.872,336.796,-153.804,170.258,52.724,160.345
C00632=1011.865,336.548,-153.770,170.250,52.729,160.344
C00633=1011.859,336.301,-153.735,170.242,52.734,160.344
C00634=1011.851,336.053,-153.701,170.234,52.739,160.344
C00635=1011.846,335.806,-153.667,170.226,52.744,160.343
C00636=1011.839,335.558,-153.631,170.219,52.749,160.343
C00637=1011.832,335.310,-153.597,170.211,52.754,160.343
C00638=1011.826,335.063,-153.563,170.204,52.760,160.342
C00639=1011.820,334.816,-153.528,170.195,52.764,160.342
C00640=1011.813,334.568,-153.493,170.189,52.769,160.342
C00641=1011.807,334.321,-153.459,170.181,52.775,160.342
C00642=1011.801,334.073,-153.425,170.173,52.780,160.341
C00643=1011.794,333.825,-153.390,170.165,52.785,160.341
C00644=1011.787,333.578,-153.356,170.158,52.791,160.341
C00645=1011.781,333.330,-153.322,170.151,52.795,160.340
C00646=1011.775,333.083,-153.288,170.143,52.801,160.340
C00647=1011.769,332.835,-153.254,170.135,52.806,160.340
C00648=1011.763,332.588,-153.219,170.128,52.811,160.339
C00649=1011.756,332.340,-153.185,170.120,52.816,160.339
C00650=1011.751,332.092,-153.151,170.113,52.821,160.339
C00651=1011.744,331.844,-153.117,170.105,52.827,160.339
C00652=1011.738,331.597,-153.083,170.097,52.832,160.338
C00653=1011.731,331.349,-153.049,170.091,52.837,160.338
C00654=1011.725,331.102,-153.015,170.083,52.843,160.338
C00655=1011.718,330.855,-152.981,170.075,52.848,160.337
C00656=1011.712,330.607,-152.947,170.067,52.853,160.337
C00657=1011.706,330.359,-152.912,170.061,52.858,160.337
C00658=1011.699,330.112,-152.880,170.053,52.864,160.337
C00659=1011.693,329.864,-152.845,170.045,52.869,160.337
C00660=1011.687,329.616,-152.811,170.038,52.875,160.336
C00661=1011.680,329.369,-152.778,170.031,52.880,160.336
C00662=1011.674,329.121,-152.744,170.023,52.885,160.336
C00663=1011.668,328.874,-152.710,170.016,52.891,160.336
C00664=1011.661,328.626,-152.676,170.008,52.896,160.335
C00665=1011.656,328.378,-152.643,170.001,52.901,160.335
C00666=1011.649,328.131,-152.609,169.994,52.907,160.335
C00667=1011.643,327.882,-152.576,169.986,52.913,160.335
C00668=1011.637,327.635,-152.542,169.979,52.918,160.335
C00669=1011.630,327.388,-152.508,169.972,52.924,160.335
C00670=1011.625,327.140,-152.475,169.964,52.929,160.334
C00671=1011.618,326.892,-152.440,169.957,52.935,160.334
C00672=1011.612,326.645,-152.408,169.950,52.940,160.334
C00673=1011.606,326.397,-152.374,169.942,52.945,160.334
C00674=1011.601,326.149,-152.340,169.935,52.951,160.334
C00675=1011.594,325.901,-152.307,169.929,52.956,160.333
C00676=1011.588,325.654,-152.273,169.921,52.962,160.333
C00677=1011.582,325.406,-152.240,169.913,52.967,160.333
C00678=1011.576,325.158,-152.207,169.906,52.973,160.333
C00679=1011.569,324.911,-152.173,169.899,52.979,160.333
C00680=1011.563,324.663,-152.140,169.892,52.984,160.332
C00681=1011.556,324.415,-152.108,169.885,52.990,160.332
C00682=1011.550,324.168,-152.075,169.877,52.996,160.332
C00683=1011.543,323.853,-152.033,169.868,53.003,160.332
C00684=1011.535,323.539,-151.991,169.859,53.010,160.332
C00685=1011.526,323.226,-151.949,169.850,53.017,160.332
C00686=1011.519,322.912,-151.908,169.841,53.025,160.332
C00687=1011.513,322.664,-151.875,169.833,53.030,160.331
C00688=1011.506,322.417,-151.842,169.827,53.036,160.332
C00689=1011.500,322.168,-151.809,169.819,53.042,160.331
C00690=1011.494,321.920,-151.776,169.812,53.048,160.331
C00691=1011.488,321.672,-151.744,169.806,53.053,160.331
C00692=1011.482,321.425,-151.711,169.798,53.059,160.331
C00693=1011.475,321.177,-151.678,169.791,53.065,160.331
C00694=1011.470,320.929,-151.645,169.783,53.071,160.331
C00695=1011.463,320.682,-151.612,169.777,53.077,160.331
C00696=1011.457,320.433,-151.580,169.770,53.082,160.331
C00697=1011.451,320.186,-151.547,169.762,53.088,160.330
C00698=1011.445,319.938,-151.515,169.756,53.094,160.331
C00699=1011.439,319.691,-151.482,169.749,53.100,160.330
C00700=1011.434,319.443,-151.450,169.741,53.106,160.330
C00701=1011.428,319.195,-151.417,169.735,53.111,160.330
C00702=1011.421,318.948,-151.384,169.727,53.117,160.330
C00703=1011.415,318.699,-151.352,169.720,53.123,160.330
C00704=1011.409,318.452,-151.319,169.714,53.129,160.330
C00705=1011.403,318.204,-151.287,169.707,53.135,160.330
C00706=1011.397,317.956,-151.254,169.699,53.141,160.330
C00707=1011.392,317.709,-151.222,169.692,53.147,160.330
C00708=1011.386,317.460,-151.190,169.686,53.153,160.330
C00709=1011.380,317.213,-151.157,169.679,53.159,160.330
C00710=1011.374,316.965,-151.125,169.671,53.165,160.330
C00711=1011.368,316.717,-151.092,169.665,53.170,160.330
C00712=1011.363,316.469,-151.060,169.657,53.176,160.329
C00713=1011.356,316.222,-151.027,169.651,53.182,160.330
C00714=1011.350,315.973,-150.995,169.644,53.188,160.330
C00715=1011.344,315.726,-150.962,169.637,53.194,160.329
C00716=1011.339,315.478,-150.931,169.631,53.200,160.330
C00717=1011.333,315.230,-150.897,169.624,53.206,160.329
C00718=1011.327,314.982,-150.865,169.616,53.213,160.329
C00719=1011.322,314.735,-150.834,169.610,53.218,160.330
C00720=1011.315,314.487,-150.801,169.603,53.225,160.329
C00721=1011.309,314.239,-150.769,169.596,53.231,160.329
C00722=1011.304,313.991,-150.737,169.590,53.237,160.329
C00723=1011.298,313.744,-150.704,169.582,53.243,160.329
C00724=1011.292,313.495,-150.672,169.575,53.249,160.329
C00725=1011.287,313.248,-150.640,169.569,53.255,160.329
C00726=1011.281,313.000,-150.608,169.562,53.261,160.329
C00727=1011.275,312.753,-150.576,169.556,53.267,160.329
C00728=1011.269,312.504,-150.544,169.548,53.273,160.329
C00729=1011.265,312.257,-150.512,169.541,53.279,160.329
C00730=1011.259,312.008,-150.480,169.535,53.285,160.329
C00731=1011.253,311.761,-150.448,169.528,53.291,160.329
C00732=1011.247,311.513,-150.415,169.521,53.298,160.329
C00733=1011.242,311.266,-150.383,169.514,53.303,160.329
C00734=1011.236,311.018,-150.351,169.507,53.310,160.329
C00735=1011.231,310.770,-150.319,169.501,53.316,160.330
C00736=1011.225,310.522,-150.287,169.494,53.322,160.330
C00737=1011.220,310.274,-150.255,169.487,53.328,160.329
C00738=1011.214,310.026,-150.223,169.481,53.334,160.330
C00739=1011.208,309.778,-150.192,169.474,53.341,160.329
C00740=1011.203,309.531,-150.160,169.468,53.347,160.330
C00741=1011.198,309.282,-150.128,169.461,53.353,160.330
C00742=1011.192,309.035,-150.096,169.453,53.359,160.330
C00743=1011.186,308.726,-150.056,169.446,53.367,160.330
C00744=1011.178,308.417,-150.017,169.437,53.375,160.330
C00745=1011.170,308.109,-149.978,169.429,53.383,160.330
C00746=1011.163,307.801,-149.940,169.420,53.391,160.330
C00747=1011.157,307.553,-149.909,169.415,53.398,160.330
C00748=1011.152,307.305,-149.878,169.408,53.404,160.330
C00749=1011.145,307.057,-149.847,169.400,53.410,160.330
C00750=1011.140,306.809,-149.816,169.395,53.417,160.331
C00751=1011.134,306.561,-149.784,169.387,53.423,160.330
C00752=1011.129,306.313,-149.753,169.381,53.430,160.331
C00753=1011.123,306.066,-149.722,169.375,53.436,160.331
C00754=1011.117,305.817,-149.691,169.368,53.442,160.331
C00755=1011.112,305.569,-149.660,169.361,53.449,160.331
C00756=1011.106,305.322,-149.629,169.355,53.455,160.331
C00757=1011.100,305.073,-149.597,169.348,53.462,160.331
C00758=1011.094,304.826,-149.566,169.341,53.468,160.331
C00759=1011.089,304.578,-149.535,169.335,53.475,160.331
C00760=1011.083,304.330,-149.505,169.329,53.482,160.332
C00761=1011.077,304.081,-149.474,169.321,53.488,160.332
C00762=1011.071,303.834,-149.443,169.316,53.494,160.332
C00763=1011.066,303.586,-149.412,169.309,53.501,160.332
C00764=1011.060,303.338,-149.381,169.302,53.508,160.332
C00765=1011.055,303.090,-149.350,169.296,53.514,160.332
C00766=1011.048,302.842,-149.319,169.289,53.521,160.332
C00767=1011.043,302.594,-149.288,169.282,53.527,160.332
C00768=1011.037,302.346,-149.258,169.276,53.534,160.333
C00769=1011.032,302.098,-149.227,169.270,53.541,160.333
C00770=1011.027,301.850,-149.196,169.263,53.547,160.333
C00771=1011.021,301.602,-149.166,169.257,53.554,160.333
C00772=1011.016,301.354,-149.135,169.250,53.560,160.333
C00773=1011.010,301.105,-149.104,169.244,53.567,160.333
C00774=1011.004,300.858,-149.073,169.238,53.574,160.334
C00775=1010.999,300.610,-149.042,169.230,53.580,160.334
C00776=1010.993,300.362,-149.012,169.225,53.587,160.334
C00777=1010.988,300.114,-148.981,169.218,53.594,160.334
C00778=1010.982,299.866,-148.950,169.211,53.601,160.334
C00779=1010.977,299.618,-148.919,169.206,53.607,160.334
C00780=1010.971,299.370,-148.889,169.199,53.614,160.335
C00781=1010.966,299.121,-148.859,169.193,53.621,160.335
C00782=1010.961,298.873,-148.828,169.186,53.627,160.335
C00783=1010.955,298.625,-148.797,169.179,53.634,160.335
C00784=1010.950,298.377,-148.767,169.174,53.640,160.335
C00785=1010.945,298.129,-148.736,169.167,53.647,160.335
C00786=1010.939,297.882,-148.706,169.160,53.654,160.336
C00787=1010.934,297.633,-148.675,169.154,53.661,160.336
C00788=1010.928,297.386,-148.644,169.148,53.668,160.336
C00789=1010.923,297.137,-148.614,169.142,53.674,160.336
C00790=1010.918,296.890,-148.584,169.135,53.681,160.336
C00791=1010.913,296.642,-148.553,169.129,53.688,160.337
C00792=1010.908,296.393,-148.522,169.123,53.695,160.337
C00793=1010.902,296.146,-148.492,169.116,53.702,160.337
C00794=1010.897,295.897,-148.462,169.110,53.708,160.337
C00795=1010.891,295.649,-148.431,169.104,53.715,160.337
C00796=1010.886,295.401,-148.400,169.097,53.722,160.338
C00797=1010.881,295.152,-148.371,169.091,53.729,160.338
C00798=1010.876,294.905,-148.340,169.085,53.736,160.338
C00799=1010.870,294.657,-148.310,169.079,53.742,160.338
C00800=1010.866,294.408,-148.280,169.073,53.750,160.339
C00801=1010.860,294.161,-148.249,169.066,53.757,160.339
C00802=1010.855,293.912,-148.219,169.060,53.763,160.339
C00803=1010.849,293.622,-148.184,169.053,53.771,160.339
C00804=1010.843,293.332,-148.149,169.046,53.779,160.340
C00805=1010.837,293.042,-148.114,169.039,53.787,160.340
C00806=1010.831,292.751,-148.078,169.030,53.796,160.340
C00807=1010.826,292.503,-148.048,169.025,53.802,160.340
C00808=1010.821,292.255,-148.017,169.018,53.810,160.341
C00809=1010.815,292.007,-147.987,169.013,53.817,160.341
C00810=1010.810,291.759,-147.958,169.006,53.824,160.341
C00811=1010.805,291.511,-147.928,168.999,53.830,160.341
C00812=1010.800,291.263,-147.897,168.994,53.838,160.342
C00813=1010.795,291.015,-147.868,168.987,53.845,160.342
C00814=1010.789,290.766,-147.838,168.981,53.852,160.342
C00815=1010.780,290.378,-147.792,168.972,53.863,160.343
C00816=1010.772,289.989,-147.746,168.962,53.874,160.343
C00817=1010.764,289.601,-147.699,168.953,53.885,160.344
C00818=1010.755,289.213,-147.653,168.942,53.896,160.344
C00819=1010.521,290.405,-148.159,168.947,53.927,160.352
C00820=1010.529,290.748,-148.200,168.955,53.917,160.351
C00821=1010.536,291.092,-148.241,168.964,53.907,160.351
C00822=1010.543,291.437,-148.283,168.972,53.897,160.350
C00823=1010.550,291.780,-148.324,168.981,53.887,160.350
C00824=1010.555,292.028,-148.354,168.987,53.880,160.350
C00825=1010.561,292.276,-148.384,168.993,53.874,160.350
C00826=1010.566,292.525,-148.414,168.999,53.866,160.349
C00827=1010.571,292.772,-148.444,169.006,53.859,160.349
C00828=1010.577,293.065,-148.479,169.013,53.851,160.349
C00829=1010.582,293.358,-148.516,169.020,53.843,160.349
C00830=1010.589,293.650,-148.551,169.028,53.835,160.348
C00831=1010.595,293.943,-148.586,169.035,53.827,160.348
C00832=1010.600,294.191,-148.617,169.042,53.820,160.348
C00833=1010.605,294.439,-148.648,169.047,53.814,160.348
C00834=1010.610,294.687,-148.677,169.054,53.807,160.348
C00835=1010.615,294.935,-148.708,169.061,53.800,160.347
C00836=1010.621,295.184,-148.738,169.066,53.793,160.347
C00837=1010.626,295.432,-148.769,169.073,53.785,160.347
C00838=1010.632,295.679,-148.799,169.079,53.778,160.347
C00839=1010.636,295.928,-148.829,169.085,53.772,160.346
C00840=1010.642,296.175,-148.859,169.092,53.765,160.346
C00841=1010.647,296.423,-148.890,169.097,53.758,160.346
C00842=1010.652,296.672,-148.920,169.104,53.751,160.346
C00843=1010.658,296.920,-148.951,169.111,53.744,160.346
C00844=1010.663,297.168,-148.981,169.116,53.738,160.345
C00845=1010.668,297.416,-149.012,169.123,53.731,160.345
C00846=1010.673,297.664,-149.041,169.130,53.725,160.345
C00847=1010.678,297.912,-149.072,169.136,53.718,160.345
C00848=1010.684,298.160,-149.103,169.143,53.711,160.345
C00849=1010.689,298.408,-149.133,169.148,53.705,160.345
C00850=1010.694,298.656,-149.164,169.155,53.698,160.344
C00851=1010.700,298.904,-149.194,169.162,53.691,160.344
C00852=1010.705,299.153,-149.225,169.168,53.684,160.344
C00853=1010.711,299.400,-149.255,169.174,53.677,160.344
C00854=1010.716,299.648,-149.286,169.181,53.670,160.344
C00855=1010.722,299.896,-149.317,169.187,53.664,160.344
C00856=1010.727,300.144,-149.348,169.194,53.657,160.344
C00857=1010.733,300.392,-149.378,169.201,53.651,160.343
C00858=1010.738,300.640,-149.409,169.206,53.644,160.343
C00859=1010.744,300.888,-149.439,169.213,53.637,160.343
C00860=1010.749,301.136,-149.470,169.220,53.631,160.343
C00861=1010.754,301.384,-149.501,169.226,53.624,160.343
C00862=1010.759,301.632,-149.531,169.233,53.617,160.343
C00863=1010.765,301.880,-149.562,169.238,53.611,160.342
C00864=1010.771,302.129,-149.593,169.245,53.605,160.342
C00865=1010.777,302.377,-149.623,169.252,53.598,160.342
C00866=1010.782,302.625,-149.654,169.258,53.591,160.342
C00867=1010.788,302.873,-149.685,169.265,53.584,160.342
C00868=1010.793,303.120,-149.716,169.272,53.578,160.342
C00869=1010.799,303.368,-149.747,169.277,53.571,160.342
C00870=1010.804,303.616,-149.778,169.284,53.564,160.341
C00871=1010.810,303.865,-149.808,169.291,53.558,160.341
C00872=1010.815,304.113,-149.839,169.297,53.552,160.341
C00873=1010.822,304.360,-149.870,169.304,53.545,160.341
C00874=1010.827,304.608,-149.901,169.311,53.538,160.341
C00875=1010.832,304.856,-149.932,169.317,53.532,160.341
C00876=1010.838,305.105,-149.963,169.324,53.526,160.341
C00877=1010.844,305.352,-149.994,169.331,53.519,160.341
C00878=1010.849,305.600,-150.025,169.338,53.513,160.341
C00879=1010.855,305.848,-150.055,169.344,53.506,160.340
C00880=1010.861,306.096,-150.087,169.351,53.500,160.341
C00881=1010.867,306.344,-150.118,169.357,53.493,160.340
C00882=1010.872,306.592,-150.149,169.364,53.487,160.340
C00883=1010.879,306.840,-150.180,169.370,53.480,160.340
C00884=1010.884,307.088,-150.211,169.378,53.474,160.340
C00885=1010.890,307.335,-150.242,169.383,53.467,160.340
C00886=1010.896,307.584,-150.274,169.390,53.461,160.340
C00887=1010.902,307.831,-150.305,169.397,53.454,160.340
C00888=1010.909,308.142,-150.344,169.406,53.447,160.340
C00889=1010.916,308.453,-150.383,169.413,53.439,160.340
C00890=1010.923,308.763,-150.422,169.422,53.431,160.340
C00891=1010.930,309.074,-150.462,169.430,53.423,160.339
C00892=1010.936,309.323,-150.494,169.437,53.416,160.340
C00893=1010.941,309.570,-150.526,169.444,53.410,160.339
C00894=1010.947,309.819,-150.558,169.451,53.404,160.340
C00895=1010.952,310.066,-150.589,169.457,53.397,160.339
C00896=1010.957,310.314,-150.621,169.464,53.392,160.339
C00897=1010.963,310.562,-150.653,169.471,53.385,160.339
C00898=1010.969,310.809,-150.685,169.478,53.379,160.339
C00899=1010.974,311.058,-150.717,169.484,53.373,160.339
C00900=1010.979,311.305,-150.749,169.491,53.367,160.339
C00901=1010.985,311.553,-150.781,169.497,53.361,160.339
C00902=1010.991,311.801,-150.813,169.504,53.354,160.339
C00903=1010.996,312.049,-150.844,169.512,53.348,160.339
C00904=1011.002,312.297,-150.876,169.518,53.342,160.339
C00905=1011.007,312.544,-150.909,169.525,53.336,160.339
C00906=1011.013,312.792,-150.941,169.532,53.330,160.339
C00907=1011.018,313.040,-150.973,169.538,53.324,160.339
C00908=1011.024,313.288,-151.005,169.545,53.318,160.339
C00909=1011.030,313.536,-151.037,169.553,53.312,160.339
C00910=1011.036,313.783,-151.070,169.559,53.306,160.339
C00911=1011.041,314.032,-151.102,169.566,53.300,160.339
C00912=1011.047,314.279,-151.134,169.572,53.294,160.339
C00913=1011.053,314.527,-151.166,169.579,53.288,160.339
C00914=1011.059,314.775,-151.199,169.587,53.281,160.339
C00915=1011.064,315.022,-151.230,169.593,53.276,160.339
C00916=1011.070,315.271,-151.262,169.600,53.269,160.339
C00917=1011.075,315.518,-151.295,169.607,53.263,160.339
C00918=1011.081,315.766,-151.327,169.613,53.257,160.339
C00919=1011.087,316.014,-151.359,169.621,53.251,160.339
C00920=1011.094,316.262,-151.392,169.628,53.246,160.340
C00921=1011.099,316.509,-151.424,169.635,53.239,160.340
C00922=1011.105,316.757,-151.456,169.642,53.234,160.340
C00923=1011.110,317.005,-151.489,169.649,53.227,160.340
C00924=1011.117,317.253,-151.522,169.656,53.221,160.340
C00925=1011.122,317.501,-151.554,169.662,53.215,160.340
C00926=1011.128,317.748,-151.586,169.670,53.210,160.340
C00927=1011.134,317.996,-151.618,169.677,53.204,160.340
C00928=1011.141,318.244,-151.651,169.683,53.198,160.340
C00929=1011.145,318.492,-151.683,169.691,53.192,160.340
C00930=1011.152,318.739,-151.716,169.698,53.186,160.340
C00931=1011.158,318.987,-151.749,169.704,53.180,160.340
C00932=1011.164,319.235,-151.781,169.712,53.174,160.340
C00933=1011.170,319.483,-151.814,169.719,53.168,160.340
C00934=1011.176,319.731,-151.847,169.726,53.162,160.341
C00935=1011.182,319.979,-151.879,169.733,53.157,160.341
C00936=1011.188,320.227,-151.912,169.740,53.151,160.341
C00937=1011.194,320.474,-151.944,169.747,53.145,160.341
C00938=1011.200,320.722,-151.976,169.754,53.139,160.341
C00939=1011.206,320.969,-152.009,169.761,53.134,160.341
C00940=1011.212,321.217,-152.042,169.769,53.127,160.341
C00941=1011.218,321.465,-152.075,169.776,53.122,160.341
C00942=1011.224,321.712,-152.108,169.782,53.116,160.341
C00943=1011.230,321.961,-152.140,169.790,53.110,160.341
C00944=1011.236,322.208,-152.172,169.797,53.104,160.342
C00945=1011.243,322.457,-152.206,169.804,53.098,160.342
C00946=1011.249,322.704,-152.239,169.811,53.093,160.342
C00947=1011.255,322.952,-152.272,169.818,53.087,160.342
C00948=1011.263,323.268,-152.313,169.828,53.080,160.342
C00949=1011.271,323.584,-152.355,169.837,53.073,160.342
C00950=1011.278,323.900,-152.397,169.847,53.065,160.342
C00951=1011.287,324.217,-152.440,169.856,53.058,160.343
C00952=1011.293,324.465,-152.472,169.863,53.052,160.343
C00953=1011.299,324.712,-152.505,169.870,53.047,160.343
C00954=1011.306,324.960,-152.538,169.877,53.041,160.343
C00955=1011.312,325.208,-152.571,169.884,53.035,160.343
C00956=1011.318,325.456,-152.604,169.892,53.030,160.343
C00957=1011.324,325.703,-152.638,169.899,53.025,160.344
C00958=1011.330,325.951,-152.671,169.906,53.019,160.344
C00959=1011.336,326.199,-152.704,169.914,53.013,160.344
C00960=1011.342,326.446,-152.738,169.921,53.007,160.344
C00961=1011.349,326.694,-152.771,169.928,53.002,160.344
C00962=1011.354,326.942,-152.806,169.936,52.997,160.345
C00963=1011.361,327.189,-152.838,169.943,52.991,160.345
C00964=1011.367,327.437,-152.872,169.950,52.986,160.345
C00965=1011.372,327.684,-152.906,169.957,52.980,160.345
C00966=1011.379,327.932,-152.939,169.965,52.974,160.345
C00967=1011.385,328.180,-152.973,169.972,52.969,160.346
C00968=1011.391,328.427,-153.007,169.979,52.964,160.346
C00969=1011.398,328.676,-153.040,169.987,52.958,160.346
C00970=1011.404,328.923,-153.074,169.994,52.953,160.346
C00971=1011.409,329.170,-153.108,170.002,52.947,160.346
C00972=1011.416,329.418,-153.141,170.009,52.942,160.347
C00973=1011.422,329.666,-153.175,170.016,52.937,160.347
C00974=1011.428,329.913,-153.209,170.024,52.931,160.347
C00975=1011.435,330.161,-153.242,170.032,52.926,160.347
C00976=1011.441,330.409,-153.276,170.039,52.920,160.348
C00977=1011.448,330.656,-153.310,170.046,52.915,160.348
C00978=1011.454,330.904,-153.344,170.054,52.910,160.348
C00979=1011.460,331.152,-153.378,170.061,52.904,160.348
C00980=1011.467,331.399,-153.412,170.069,52.899,160.349
C00981=1011.472,331.646,-153.446,170.077,52.894,160.349
C00982=1011.479,331.894,-153.480,170.084,52.889,160.349
C00983=1011.485,332.142,-153.514,170.091,52.883,160.349
C00984=1011.491,332.390,-153.548,170.099,52.878,160.350
C00985=1011.497,332.637,-153.583,170.107,52.872,160.350
C00986=1011.504,332.885,-153.616,170.114,52.868,160.350
C00987=1011.510,333.132,-153.650,170.122,52.862,160.351
C00988=1011.517,333.380,-153.685,170.129,52.857,160.351
C00989=1011.523,333.628,-153.719,170.137,52.852,160.351
C00990=1011.529,333.875,-153.753,170.145,52.847,160.352
C00991=1011.536,334.123,-153.788,170.152,52.842,160.352
C00992=1011.542,334.370,-153.822,170.159,52.836,160.352
C00993=1011.548,334.618,-153.857,170.167,52.831,160.352
C00994=1011.554,334.866,-153.891,170.175,52.826,160.353
C00995=1011.560,335.113,-153.925,170.183,52.821,160.353
C00996=1011.568,335.360,-153.960,170.190,52.816,160.353
C00997=1011.574,335.608,-153.994,170.198,52.810,160.353
C00998=1011.580,335.855,-154.028,170.206,52.806,160.354
C00999=1011.587,336.103,-154.064,170.213,52.800,160.354
C01000=1011.593,336.351,-154.098,170.221,52.795,160.355
C01001=1011.599,336.598,-154.132,170.229,52.790,160.355
C01002=1011.606,336.845,-154.167,170.236,52.785,160.355
C01003=1011.612,337.093,-154.202,170.244,52.780,160.356
C01004=1011.619,337.341,-154.237,170.252,52.775,160.356
C01005=1011.625,337.588,-154.271,170.260,52.770,160.356
C01006=1011.633,337.835,-154.305,170.268,52.765,160.357
C01007=1011.639,338.083,-154.340,170.276,52.760,160.357
C01008=1011.647,338.395,-154.384,170.286,52.754,160.358
C01009=1011.655,338.707,-154.428,170.295,52.748,160.358
C01010=1011.663,339.019,-154.472,170.305,52.741,160.359
C01011=1011.671,339.331,-154.516,170.315,52.735,160.359
C01012=1011.678,339.578,-154.551,170.323,52.730,160.359
C01013=1011.685,339.826,-154.585,170.330,52.725,160.360
C01014=1011.691,340.074,-154.621,170.338,52.720,160.360
C01015=1011.697,340.321,-154.656,170.347,52.715,160.361
C01016=1011.704,340.569,-154.691,170.355,52.710,160.361
C01017=1011.711,340.816,-154.727,170.362,52.706,160.361
C01018=1011.718,341.063,-154.762,170.369,52.701,160.362
C01019=1011.724,341.311,-154.797,170.378,52.696,160.362
C01020=1011.730,341.558,-154.833,170.386,52.691,160.363
C01021=1011.737,341.806,-154.868,170.394,52.686,160.363
C01022=1011.744,342.053,-154.903,170.402,52.681,160.364
C01023=1011.751,342.300,-154.938,170.410,52.677,160.364
C01024=1011.757,342.548,-154.973,170.418,52.672,160.364
C01025=1011.764,342.796,-155.009,170.426,52.667,160.365
C01026=1011.770,343.043,-155.044,170.433,52.663,160.365
C01027=1011.777,343.290,-155.079,170.441,52.658,160.366
C01028=1011.784,343.538,-155.114,170.450,52.653,160.366
C01029=1011.790,343.785,-155.150,170.458,52.648,160.367
C01030=1011.797,344.033,-155.185,170.466,52.643,160.367
C01031=1011.804,344.279,-155.221,170.474,52.639,160.368
C01032=1011.810,344.527,-155.256,170.482,52.634,160.368
C01033=1011.817,344.775,-155.292,170.490,52.629,160.368
C01034=1011.824,345.023,-155.327,170.498,52.624,160.369
C01035=1011.831,345.269,-155.363,170.507,52.620,160.370
C01036=1011.838,345.517,-155.398,170.515,52.615,160.370
C01037=1011.844,345.764,-155.434,170.523,52.610,160.371
C01038=1011.851,346.012,-155.470,170.531,52.606,160.371
C01039=1011.858,346.259,-155.505,170.539,52.601,160.371
C01040=1011.865,346.506,-155.542,170.548,52.597,160.372
C01041=1011.871,346.754,-155.577,170.555,52.592,160.373
C01042=1011.878,347.001,-155.613,170.563,52.587,160.373
C01043=1011.885,347.248,-155.650,170.572,52.583,160.374
C01044=1011.891,347.496,-155.685,170.580,52.579,160.374
C01045=1011.898,347.742,-155.721,170.588,52.574,160.375
C01046=1011.905,347.990,-155.758,170.596,52.570,160.375
C01047=1011.912,348.238,-155.793,170.604,52.565,160.376
C01048=1011.918,348.485,-155.830,170.613,52.561,160.376
C01049=1011.926,348.732,-155.866,170.621,52.556,160.377
C01050=1011.932,348.979,-155.902,170.629,52.551,160.377
C01051=1011.939,349.226,-155.937,170.638,52.547,160.378
C01052=1011.946,349.474,-155.974,170.646,52.542,160.378
C01053=1011.953,349.721,-156.010,170.654,52.538,160.379
C01054=1011.960,349.969,-156.047,170.663,52.534,160.380
C01055=1011.967,350.215,-156.083,170.671,52.529,160.380
C01056=1011.974,350.463,-156.120,170.680,52.525,160.381
C01057=1011.981,350.710,-156.155,170.688,52.520,160.381
C01058=1011.988,350.958,-156.192,170.696,52.516,160.382
C01059=1011.995,351.204,-156.228,170.705,52.512,160.383
C01060=1012.002,351.452,-156.265,170.713,52.507,160.383
C01061=1012.009,351.699,-156.301,170.721,52.503,160.384
C01062=1012.016,351.947,-156.338,170.730,52.499,160.384
C01063=1012.023,352.193,-156.373,170.739,52.494,160.385
C01064=1012.030,352.441,-156.410,170.748,52.490,160.386
C01065=1012.038,352.689,-156.446,170.756,52.485,160.386
C01066=1012.044,352.936,-156.483,170.765,52.481,160.387
C01067=1012.052,353.183,-156.520,170.773,52.476,160.387
C01068=1012.060,353.492,-156.566,170.783,52.472,160.388
C01069=1012.068,353.802,-156.611,170.795,52.466,160.389
C01070=1012.078,354.111,-156.658,170.805,52.461,160.390
C01071=1012.087,354.420,-156.704,170.816,52.456,160.391
C01072=1012.094,354.667,-156.740,170.824,52.452,160.392
C01073=1012.101,354.915,-156.777,170.833,52.448,160.392
C01074=1012.108,355.162,-156.814,170.842,52.443,160.393
C01075=1012.116,355.409,-156.851,170.851,52.439,160.394
C01076=1012.123,355.656,-156.888,170.859,52.435,160.394
C01077=1012.130,355.904,-156.925,170.868,52.431,160.395
C01078=1012.138,356.151,-156.962,170.876,52.426,160.396
C01079=1012.144,356.397,-156.999,170.885,52.422,160.396
C01080=1012.151,356.645,-157.036,170.893,52.418,160.397
C01081=1012.159,356.892,-157.073,170.902,52.414,160.398
C01082=1012.167,357.139,-157.110,170.912,52.410,160.398
C01083=1012.173,357.387,-157.147,170.920,52.405,160.399
C01084=1012.181,357.634,-157.185,170.929,52.402,160.400
C01085=1012.187,357.880,-157.222,170.938,52.398,160.401
C01086=1012.195,358.127,-157.259,170.946,52.394,160.401
C01087=1012.203,358.374,-157.296,170.955,52.390,160.402
C01088=1012.210,358.621,-157.334,170.965,52.386,160.403
C01089=1012.217,358.869,-157.371,170.973,52.382,160.404
C01090=1012.224,359.116,-157.409,170.982,52.377,160.404
C01091=1012.232,359.363,-157.446,170.991,52.374,160.405
C01092=1012.239,359.610,-157.484,170.999,52.370,160.406
C01093=1012.246,359.857,-157.521,171.008,52.366,160.407
C01094=1012.253,360.104,-157.559,171.018,52.362,160.407
C01095=1012.261,360.351,-157.596,171.027,52.358,160.408
C01096=1012.268,360.598,-157.634,171.035,52.354,160.409
C01097=1012.275,360.845,-157.672,171.044,52.351,160.410
C01098=1012.282,361.092,-157.710,171.053,52.347,160.411
C01099=1012.289,361.340,-157.748,171.063,52.343,160.412
C01100=1012.296,361.587,-157.785,171.071,52.339,160.412
C01101=1012.304,361.833,-157.824,171.080,52.335,160.413
C01102=1012.312,362.081,-157.862,171.089,52.331,160.414
C01103=1012.319,362.328,-157.900,171.099,52.327,160.415
C01104=1012.326,362.575,-157.937,171.108,52.324,160.416
C01105=1012.334,362.822,-157.975,171.116,52.319,160.416
C01106=1012.341,363.068,-158.013,171.125,52.316,160.417
C01107=1012.349,363.316,-158.051,171.135,52.312,160.418
C01108=1012.357,363.563,-158.089,171.144,52.309,160.419
C01109=1012.364,363.810,-158.127,171.153,52.304,160.420
C01110=1012.371,364.056,-158.165,171.163,52.301,160.421
C01111=1012.379,364.304,-158.203,171.172,52.297,160.422
C01112=1012.387,364.551,-158.241,171.181,52.294,160.422
C01113=1012.394,364.797,-158.279,171.191,52.290,160.423
C01114=1012.402,365.045,-158.317,171.199,52.286,160.424
C01115=1012.410,365.292,-158.356,171.208,52.282,160.425
C01116=1012.417,365.538,-158.394,171.218,52.278,160.426
C01117=1012.426,365.785,-158.432,171.227,52.275,160.427
C01118=1012.433,366.032,-158.470,171.236,52.271,160.428
C01119=1012.440,366.279,-158.508,171.246,52.267,160.429
C01120=1012.448,366.526,-158.547,171.255,52.264,160.430
C01121=1012.456,366.773,-158.585,171.264,52.260,160.430
C01122=1012.464,367.020,-158.624,171.274,52.257,160.431
C01123=1012.471,367.267,-158.662,171.283,52.253,160.432
C01124=1012.479,367.514,-158.701,171.294,52.250,160.433
C01125=1012.487,367.760,-158.739,171.302,52.246,160.434
C01126=1012.494,368.008,-158.778,171.311,52.243,160.435
C01127=1012.502,368.254,-158.817,171.321,52.239,160.436
C01128=1012.511,368.538,-158.862,171.332,52.235,160.437
C01129=1012.519,368.823,-158.907,171.343,52.231,160.438
C01130=1012.528,369.107,-158.952,171.354,52.227,160.440
C01131=1012.537,369.391,-158.996,171.365,52.224,160.441
C01132=1012.545,369.639,-159.035,171.375,52.220,160.442
C01133=1012.553,369.885,-159.074,171.384,52.216,160.443
C01134=1012.560,370.132,-159.113,171.394,52.213,160.444
C01135=1012.568,370.379,-159.152,171.403,52.209,160.445
C01136=1012.577,370.626,-159.191,171.412,52.206,160.446
C01137=1012.583,370.873,-159.230,171.423,52.203,160.447
C01138=1012.592,371.119,-159.269,171.432,52.199,160.448
C01139=1012.600,371.366,-159.308,171.442,52.196,160.449
C01140=1012.607,371.613,-159.347,171.452,52.193,160.450
C01141=1012.616,371.859,-159.387,171.462,52.189,160.451
C01142=1012.624,372.106,-159.425,171.471,52.186,160.452
C01143=1012.632,372.353,-159.465,171.481,52.183,160.453
C01144=1012.640,372.600,-159.505,171.490,52.180,160.454
C01145=1012.648,372.846,-159.543,171.501,52.176,160.455
C01146=1012.655,373.093,-159.583,171.511,52.173,160.456
C01147=1012.664,373.340,-159.622,171.520,52.170,160.457
C01148=1012.672,373.587,-159.661,171.531,52.166,160.459
C01149=1012.680,373.834,-159.701,171.539,52.163,160.459
C01150=1012.688,374.081,-159.740,171.550,52.160,160.461
C01151=1012.696,374.327,-159.779,171.559,52.157,160.462
C01152=1012.704,374.574,-159.819,171.570,52.154,160.463
C01153=1012.713,374.821,-159.859,171.580,52.150,160.464
C01154=1012.720,375.068,-159.898,171.589,52.148,160.465
C01155=1012.729,375.314,-159.938,171.600,52.144,160.466
C01156=1012.737,375.561,-159.978,171.609,52.141,160.467
C01157=1012.745,375.807,-160.018,171.620,52.138,160.469
C01158=1012.753,376.054,-160.058,171.630,52.135,160.470
C01159=1012.761,376.301,-160.098,171.639,52.132,160.471
C01160=1012.769,376.547,-160.138,171.650,52.129,160.472
C01161=1012.777,376.794,-160.178,171.660,52.126,160.473
C01162=1012.785,377.041,-160.217,171.670,52.123,160.474
C01163=1012.793,377.287,-160.258,171.680,52.119,160.476
C01164=1012.801,377.534,-160.297,171.690,52.116,160.477
C01165=1012.809,377.780,-160.338,171.700,52.114,160.478
C01166=1012.817,378.027,-160.378,171.711,52.111,160.479
C01167=1012.825,378.273,-160.419,171.721,52.107,160.480
C01168=1012.834,378.520,-160.458,171.730,52.105,160.481
C01169=1012.842,378.767,-160.499,171.741,52.102,160.483
C01170=1012.850,379.014,-160.539,171.752,52.099,160.484
C01171=1012.859,379.260,-160.579,171.762,52.096,160.485
C01172=1012.867,379.507,-160.620,171.772,52.093,160.487
C01173=1012.875,379.753,-160.660,171.782,52.090,160.488
C01174=1012.884,379.999,-160.700,171.793,52.087,160.489
C01175=1012.893,380.246,-160.741,171.803,52.084,160.490
C01176=1012.901,380.493,-160.782,171.814,52.081,160.492
C01177=1012.909,380.739,-160.822,171.824,52.079,160.493
C01178=1012.918,380.986,-160.862,171.834,52.076,160.494
C01179=1012.926,381.233,-160.902,171.845,52.073,160.495
C01180=1012.934,381.479,-160.943,171.856,52.070,160.497
C01181=1012.943,381.726,-160.984,171.866,52.067,160.498
C01182=1012.951,381.972,-161.024,171.876,52.065,160.499
C01183=1012.960,382.218,-161.065,171.887,52.062,160.501
C01184=1012.618,380.147,-161.074,171.781,52.143,160.501
C01185=1012.610,379.901,-161.033,171.770,52.146,160.500
C01186=1012.602,379.655,-160.993,171.760,52.149,160.499
C01187=1012.593,379.408,-160.953,171.750,52.151,160.497
C01188=1012.585,379.161,-160.912,171.740,52.155,160.496
C01189=1012.577,378.915,-160.872,171.729,52.157,160.495
C01190=1012.568,378.668,-160.833,171.719,52.160,160.494
C01191=1012.560,378.422,-160.792,171.708,52.164,160.493
C01192=1012.552,378.175,-160.752,171.698,52.166,160.491
C01193=1012.543,377.928,-160.712,171.688,52.169,160.490
C01194=1012.535,377.681,-160.672,171.678,52.172,160.489
C01195=1012.527,377.435,-160.631,171.668,52.175,160.488
C01196=1012.519,377.189,-160.592,171.658,52.179,160.487
C01197=1012.511,376.942,-160.552,171.647,52.181,160.485
C01198=1012.503,376.695,-160.511,171.638,52.184,160.484
C01199=1012.495,376.449,-160.472,171.627,52.187,160.483
C01200=1012.487,376.202,-160.432,171.617,52.191,160.482
C01201=1012.479,375.956,-160.391,171.607,52.193,160.481
C01202=1012.470,375.709,-160.352,171.597,52.197,160.479
C01203=1012.463,375.462,-160.312,171.587,52.200,160.478
C01204=1012.455,375.215,-160.272,171.577,52.203,160.477
C01205=1012.447,374.969,-160.233,171.567,52.206,160.476
C01206=1012.439,374.722,-160.193,171.557,52.209,160.475
C01207=1012.430,374.475,-160.154,171.547,52.212,160.474
C01208=1012.423,374.228,-160.114,171.537,52.215,160.472
C01209=1012.414,373.982,-160.074,171.528,52.219,160.471
C01210=1012.406,373.735,-160.035,171.517,52.222,160.470
C01211=1012.399,373.488,-159.996,171.507,52.225,160.469
C01212=1012.390,373.242,-159.957,171.497,52.228,160.468
C01213=1012.382,372.995,-159.917,171.487,52.232,160.467
C01214=1012.375,372.747,-159.878,171.478,52.235,160.466
C01215=1012.366,372.501,-159.839,171.468,52.238,160.465
C01216=1012.358,372.254,-159.800,171.459,52.242,160.464
C01217=1012.351,372.007,-159.761,171.448,52.245,160.463
C01218=1012.342,371.761,-159.721,171.439,52.248,160.462
C01219=1012.334,371.514,-159.682,171.429,52.252,160.461
C01220=1012.327,371.267,-159.643,171.419,52.255,160.459
C01221=1012.319,371.021,-159.604,171.410,52.259,160.459
C01222=1012.311,370.774,-159.565,171.399,52.262,160.457
C01223=1012.303,370.526,-159.526,171.390,52.265,160.456
C01224=1012.295,370.280,-159.487,171.380,52.269,160.455
C01225=1012.288,370.035,-159.449,171.371,52.272,160.454
C01226=1012.280,369.791,-159.410,171.362,52.276,160.453
C01227=1012.272,369.546,-159.371,171.351,52.279,160.452
C01228=1012.264,369.301,-159.333,171.342,52.282,160.451
C01229=1012.257,369.057,-159.294,171.333,52.286,160.451
C01230=1012.249,368.812,-159.256,171.323,52.289,160.449
C01231=1012.242,368.568,-159.217,171.314,52.293,160.448
C01232=1012.234,368.323,-159.179,171.305,52.296,160.448
C01233=1012.226,368.076,-159.141,171.295,52.300,160.447
C01234=1012.219,367.829,-159.102,171.286,52.303,160.445
C01235=1012.211,367.582,-159.063,171.276,52.307,160.444
C01236=1012.203,367.335,-159.025,171.267,52.310,160.444
C01237=1012.196,367.088,-158.986,171.258,52.314,160.443
C01238=1012.189,366.842,-158.948,171.248,52.318,160.442
C01239=1012.181,366.594,-158.909,171.239,52.321,160.441
C01240=1012.173,366.348,-158.871,171.229,52.325,160.440
C01241=1012.165,366.101,-158.832,171.220,52.328,160.439
C01242=1012.157,365.854,-158.794,171.211,52.332,160.438
C01243=1012.151,365.607,-158.756,171.201,52.336,160.437
C01244=1012.143,365.359,-158.717,171.192,52.339,160.436
C01245=1012.135,365.113,-158.679,171.182,52.343,160.435
C01246=1012.128,364.866,-158.641,171.173,52.347,160.434
C01247=1012.120,364.619,-158.603,171.164,52.350,160.433
C01248=1012.112,364.372,-158.565,171.154,52.354,160.432
C01249=1012.105,364.125,-158.527,171.145,52.358,160.432
C01250=1012.098,363.878,-158.489,171.137,52.362,160.431
C01251=1012.090,363.631,-158.451,171.127,52.366,160.430
C01252=1012.082,363.384,-158.413,171.118,52.369,160.429
C01253=1012.075,363.137,-158.375,171.109,52.373,160.428
C01254=1012.067,362.890,-158.337,171.100,52.377,160.428
C01255=1012.060,362.643,-158.299,171.090,52.381,160.427
C01256=1012.052,362.395,-158.262,171.081,52.384,160.426
C01257=1012.045,362.149,-158.223,171.073,52.388,160.425
C01258=1012.037,361.902,-158.186,171.063,52.392,160.424
C01259=1012.030,361.655,-158.148,171.054,52.396,160.423
C01260=1012.023,361.408,-158.110,171.045,52.400,160.422
C01261=1012.015,361.161,-158.072,171.036,52.403,160.422
C01262=1012.008,360.914,-158.035,171.027,52.408,160.421
C01263=1012.001,360.667,-157.997,171.018,52.411,160.420
C01264=1011.994,360.420,-157.960,171.009,52.415,160.419
C01265=1011.986,360.173,-157.922,171.000,52.419,160.418
C01266=1011.979,359.926,-157.884,170.991,52.423,160.418
C01267=1011.972,359.679,-157.847,170.982,52.428,160.417
C01268=1011.964,359.432,-157.809,170.973,52.431,160.416
C01269=1011.957,359.185,-157.772,170.965,52.435,160.415
C01270=1011.950,358.937,-157.734,170.956,52.439,160.414
C01271=1011.943,358.690,-157.696,170.946,52.443,160.414
C01272=1011.935,358.443,-157.659,170.937,52.447,160.413
C01273=1011.928,358.196,-157.621,170.928,52.451,160.412
C01274=1011.922,357.949,-157.585,170.920,52.455,160.411
C01275=1011.914,357.702,-157.548,170.911,52.459,160.411
C01276=1011.907,357.455,-157.511,170.903,52.463,160.410
C01277=1011.899,357.208,-157.473,170.893,52.468,160.409
C01278=1011.892,356.960,-157.436,170.884,52.471,160.408
C01279=1011.884,356.713,-157.399,170.876,52.475,160.408
C01280=1011.878,356.467,-157.362,170.867,52.480,160.407
C01281=1011.871,356.219,-157.325,170.859,52.484,160.406
C01282=1011.864,355.972,-157.288,170.850,52.488,160.406
C01283=1011.856,355.725,-157.252,170.841,52.492,160.405
C01284=1011.849,355.477,-157.214,170.832,52.497,160.404
C01285=1011.842,355.230,-157.178,170.823,52.501,160.404
C01286=1011.834,354.984,-157.141,170.815,52.505,160.403
C01287=1011.827,354.736,-157.104,170.806,52.509,160.402
C01288=1011.821,354.489,-157.067,170.798,52.513,160.402
C01289=1011.811,354.177,-157.020,170.786,52.518,160.401
C01290=1011.803,353.865,-156.974,170.776,52.524,160.400
C01291=1011.794,353.553,-156.928,170.765,52.529,160.399
C01292=1011.785,353.242,-156.882,170.755,52.535,160.398
C01293=1011.778,352.995,-156.845,170.746,52.539,160.398
C01294=1011.771,352.748,-156.808,170.737,52.543,160.397
C01295=1011.764,352.500,-156.772,170.729,52.547,160.396
C01296=1011.757,352.253,-156.736,170.720,52.553,160.396
C01297=1011.750,352.006,-156.700,170.711,52.557,160.395
C01298=1011.743,351.759,-156.663,170.703,52.561,160.394
C01299=1011.736,351.511,-156.627,170.694,52.565,160.394
C01300=1011.729,351.264,-156.590,170.686,52.570,160.393
C01301=1011.722,351.017,-156.554,170.678,52.574,160.393
C01302=1011.715,350.770,-156.518,170.669,52.579,160.392
C01303=1011.708,350.522,-156.482,170.661,52.583,160.391
C01304=1011.701,350.275,-156.445,170.652,52.587,160.391
C01305=1011.694,350.028,-156.409,170.644,52.592,160.390
C01306=1011.687,349.781,-156.372,170.636,52.596,160.390
C01307=1011.680,349.533,-156.337,170.628,52.601,160.389
C01308=1011.674,349.285,-156.301,170.619,52.605,160.389
C01309=1011.667,349.039,-156.265,170.611,52.610,160.388
C01310=1011.660,348.791,-156.228,170.602,52.614,160.387
C01311=1011.653,348.544,-156.193,170.594,52.619,160.387
C01312=1011.646,348.297,-156.156,170.586,52.623,160.386
C01313=1011.639,348.049,-156.120,170.578,52.628,160.386
C01314=1011.633,347.801,-156.084,170.569,52.632,160.385
C01315=1011.626,347.555,-156.048,170.561,52.637,160.385
C01316=1011.619,347.308,-156.012,170.553,52.641,160.384
C01317=1011.612,347.060,-155.977,170.544,52.645,160.383
C01318=1011.606,346.813,-155.940,170.536,52.650,160.383
C01319=1011.599,346.565,-155.905,170.528,52.655,160.383
C01320=1011.593,346.318,-155.869,170.520,52.660,160.382
C01321=1011.585,346.070,-155.833,170.511,52.664,160.381
C01322=1011.578,345.823,-155.797,170.503,52.669,160.381
C01323=1011.572,345.576,-155.761,170.495,52.674,160.380
C01324=1011.565,345.328,-155.726,170.487,52.678,160.380
C01325=1011.558,345.082,-155.690,170.479,52.683,160.380
C01326=1011.551,344.834,-155.655,170.470,52.687,160.379
C01327=1011.545,344.586,-155.619,170.462,52.692,160.378
C01328=1011.538,344.338,-155.584,170.454,52.697,160.378
C01329=1011.531,344.091,-155.549,170.446,52.702,160.377
C01330=1011.524,343.844,-155.513,170.438,52.707,160.377
C01331=1011.517,343.597,-155.478,170.430,52.711,160.377
C01332=1011.511,343.349,-155.442,170.422,52.716,160.376
C01333=1011.505,343.102,-155.407,170.414,52.721,160.376
C01334=1011.498,342.855,-155.372,170.406,52.726,160.375
C01335=1011.491,342.607,-155.337,170.398,52.730,160.375
C01336=1011.485,342.359,-155.301,170.390,52.735,160.374
C01337=1011.478,342.112,-155.266,170.382,52.740,160.374
C01338=1011.472,341.865,-155.231,170.374,52.745,160.373
C01339=1011.465,341.617,-155.196,170.366,52.750,160.373
C01340=1011.459,341.370,-155.160,170.358,52.754,160.372
C01341=1011.452,341.122,-155.125,170.350,52.760,160.372
C01342=1011.445,340.875,-155.090,170.342,52.765,160.372
C01343=1011.439,340.627,-155.055,170.334,52.769,160.371
C01344=1011.432,340.380,-155.020,170.326,52.774,160.371
C01345=1011.426,340.133,-154.985,170.318,52.779,160.370
C01346=1011.420,339.885,-154.950,170.311,52.784,160.370
C01347=1011.413,339.637,-154.915,170.303,52.789,160.370
C01348=1011.407,339.390,-154.880,170.295,52.794,160.369
C01349=1011.398,339.076,-154.836,170.285,52.800,160.369
C01350=1011.390,338.761,-154.791,170.275,52.807,160.368
C01351=1011.381,338.447,-154.747,170.265,52.813,160.368
C01352=1011.374,338.133,-154.703,170.255,52.819,160.367
C01353=1011.367,337.886,-154.668,170.247,52.824,160.367
C01354=1011.361,337.638,-154.634,170.239,52.830,160.367
C01355=1011.354,337.390,-154.598,170.231,52.834,160.366
C01356=1011.348,337.143,-154.564,170.224,52.840,160.366
C01357=1011.342,336.895,-154.530,170.216,52.845,160.365
C01358=1011.335,336.648,-154.495,170.208,52.849,160.365
C01359=1011.328,336.400,-154.461,170.201,52.855,160.365
C01360=1011.322,336.153,-154.427,170.193,52.860,160.365
C01361=1011.315,335.905,-154.392,170.185,52.865,160.364
C01362=1011.309,335.657,-154.357,170.177,52.870,160.364
C01363=1011.303,335.410,-154.323,170.169,52.875,160.363
C01364=1011.296,335.162,-154.289,170.162,52.881,160.363
C01365=1011.290,334.916,-154.254,170.155,52.885,160.363
C01366=1011.284,334.668,-154.220,170.147,52.891,160.362
C01367=1011.277,334.420,-154.185,170.139,52.896,160.362
C01368=1011.271,334.172,-154.151,170.131,52.901,160.362
C01369=1011.264,333.925,-154.117,170.123,52.906,160.361
C01370=1011.258,333.677,-154.083,170.116,52.912,160.361
C01371=1011.252,333.429,-154.049,170.109,52.916,160.361
C01372=1011.246,333.182,-154.015,170.101,52.922,160.361
C01373=1011.239,332.934,-153.980,170.093,52.927,160.360
C01374=1011.234,332.687,-153.946,170.086,52.933,160.360
C01375=1011.227,332.439,-153.912,170.078,52.938,160.360
C01376=1011.221,332.191,-153.878,170.071,52.943,160.359
C01377=1011.215,331.943,-153.844,170.063,52.948,160.359
C01378=1011.209,331.696,-153.809,170.056,52.954,160.359
C01379=1011.202,331.449,-153.776,170.048,52.959,160.359
C01380=1011.196,331.201,-153.742,170.040,52.964,160.358
C01381=1011.190,330.954,-153.708,170.033,52.969,160.358
C01382=1011.183,330.706,-153.674,170.026,52.975,160.358
C01383=1011.177,330.458,-153.640,170.018,52.980,160.358
C01384=1011.170,330.211,-153.607,170.010,52.986,160.357
C01385=1011.164,329.963,-153.573,170.003,52.991,160.357
C01386=1011.159,329.716,-153.539,169.996,52.996,160.357
C01387=1011.151,329.468,-153.505,169.988,53.002,160.357
C01388=1011.146,329.220,-153.472,169.981,53.007,160.356
C01389=1011.140,328.973,-153.438,169.973,53.013,160.356
C01390=1011.133,328.724,-153.405,169.965,53.018,160.356
C01391=1011.127,328.477,-153.371,169.959,53.023,160.356
C01392=1011.121,328.230,-153.337,169.951,53.029,160.355
C01393=1011.115,327.982,-153.304,169.943,53.034,160.355
C01394=1011.109,327.734,-153.270,169.936,53.040,160.355
C01395=1011.102,327.487,-153.237,169.929,53.046,160.355
C01396=1011.097,327.239,-153.204,169.922,53.051,160.355
C01397=1011.091,326.991,-153.169,169.914,53.057,160.354
C01398=1011.084,326.743,-153.136,169.906,53.062,160.354
C01399=1011.078,326.496,-153.102,169.899,53.068,160.354
C01400=1011.073,326.248,-153.069,169.892,53.073,160.354
C01401=1011.066,326.000,-153.036,169.885,53.079,160.354
C01402=1011.060,325.753,-153.002,169.877,53.085,160.353
C01403=1011.055,325.505,-152.969,169.870,53.090,160.353
C01404=1011.049,325.258,-152.936,169.863,53.095,160.353
C01405=1011.042,325.009,-152.903,169.856,53.101,160.353
C01406=1011.035,324.762,-152.870,169.848,53.107,160.353
C01407=1011.030,324.514,-152.837,169.840,53.112,160.352
C01408=1011.024,324.266,-152.804,169.834,53.118,160.353
C01409=1011.016,323.948,-152.762,169.824,53.126,160.352
C01410=1011.008,323.629,-152.719,169.815,53.133,160.352
C01411=1010.999,323.311,-152.677,169.806,53.140,160.352
C01412=1010.992,322.992,-152.635,169.796,53.147,160.352
C01413=1010.985,322.744,-152.603,169.790,53.153,160.352
C01414=1010.980,322.496,-152.569,169.782,53.159,160.351
C01415=1010.973,322.249,-152.537,169.775,53.165,160.351
C01416=1010.967,322.001,-152.504,169.767,53.170,160.351
C01417=1010.961,321.753,-152.472,169.761,53.176,160.351
C01418=1010.955,321.505,-152.439,169.754,53.182,160.351
C01419=1010.949,321.258,-152.406,169.746,53.188,160.351
C01420=1010.943,321.010,-152.373,169.739,53.194,160.351
C01421=1010.937,320.762,-152.341,169.732,53.199,160.351
C01422=1010.931,320.514,-152.308,169.725,53.206,160.351
C01423=1010.924,320.267,-152.275,169.717,53.211,160.350
C01424=1010.918,320.018,-152.243,169.710,53.217,160.350
C01425=1010.913,319.771,-152.211,169.704,53.223,160.350
C01426=1010.907,319.524,-152.178,169.696,53.229,160.350
C01427=1010.901,319.275,-152.146,169.689,53.235,160.350
C01428=1010.895,319.028,-152.113,169.682,53.241,160.350
C01429=1010.889,318.780,-152.081,169.675,53.246,160.350
C01430=1010.883,318.532,-152.048,169.668,53.252,160.350
C01431=1010.878,318.284,-152.016,169.661,53.259,160.350
C01432=1010.872,318.037,-151.983,169.655,53.264,160.350
C01433=1010.866,317.788,-151.951,169.647,53.270,160.349
C01434=1010.859,317.541,-151.918,169.640,53.276,160.349
C01435=1010.854,317.293,-151.887,169.633,53.282,160.349
C01436=1010.848,317.046,-151.854,169.627,53.288,160.349
C01437=1010.842,316.797,-151.821,169.619,53.294,160.349
C01438=1010.836,316.550,-151.789,169.612,53.300,160.349
C01439=1010.831,316.302,-151.757,169.605,53.306,160.349
C01440=1010.825,316.054,-151.725,169.598,53.312,160.349
C01441=1010.819,315.806,-151.692,169.591,53.318,160.349
C01442=1010.814,315.558,-151.660,169.585,53.324,160.349
C01443=1010.808,315.310,-151.628,169.578,53.330,160.349
C01444=1010.802,315.063,-151.595,169.571,53.336,160.349
C01445=1010.796,314.815,-151.564,169.563,53.343,160.349
C01446=1010.790,314.567,-151.532,169.557,53.348,160.349
C01447=1010.785,314.319,-151.500,169.550,53.355,160.349
C01448=1010.779,314.071,-151.467,169.543,53.361,160.349
C01449=1010.774,313.824,-151.435,169.537,53.367,160.349
C01450=1010.768,313.576,-151.403,169.529,53.373,160.349
C01451=1010.762,313.327,-151.371,169.522,53.379,160.349
C01452=1010.757,313.080,-151.339,169.516,53.385,160.349
C01453=1010.751,312.832,-151.307,169.509,53.391,160.349
C01454=1010.746,312.585,-151.274,169.502,53.397,160.349
C01455=1010.740,312.337,-151.243,169.495,53.403,160.349
C01456=1010.734,312.089,-151.210,169.488,53.409,160.349
C01457=1010.729,311.841,-151.179,169.481,53.416,160.349
C01458=1010.723,311.593,-151.147,169.475,53.421,160.349
C01459=1010.717,311.346,-151.115,169.468,53.428,160.349
C01460=1010.711,311.097,-151.083,169.460,53.434,160.349
C01461=1010.707,310.850,-151.051,169.455,53.440,160.349
C01462=1010.701,310.602,-151.019,169.448,53.447,160.349
C01463=1010.695,310.354,-150.987,169.441,53.453,160.349
C01464=1010.690,310.106,-150.955,169.434,53.459,160.349
C01465=1010.684,309.858,-150.923,169.427,53.465,160.349
C01466=1010.679,309.611,-150.892,169.421,53.471,160.349
C01467=1010.674,309.362,-150.860,169.414,53.478,160.349
C01468=1010.668,309.114,-150.828,169.407,53.484,160.349
C01469=1010.661,308.802,-150.788,169.398,53.492,160.349
C01470=1010.655,308.488,-150.748,169.390,53.500,160.349
C01471=1010.647,308.176,-150.709,169.381,53.508,160.349
C01472=1010.640,307.863,-150.670,169.373,53.516,160.349
C01473=1010.634,307.614,-150.639,169.367,53.522,160.349
C01474=1010.628,307.367,-150.608,169.360,53.529,160.349
C01475=1010.623,307.118,-150.577,169.353,53.535,160.349
C01476=1010.617,306.871,-150.546,169.347,53.542,160.350
C01477=1010.611,306.623,-150.515,169.340,53.548,160.349
C01478=1010.605,306.375,-150.484,169.333,53.555,160.350
C01479=1010.600,306.126,-150.453,169.327,53.561,160.350
C01480=1010.594,305.879,-150.422,169.320,53.568,160.350
C01481=1010.589,305.631,-150.391,169.313,53.574,160.350
C01482=1010.582,305.383,-150.360,169.306,53.581,160.350
C01483=1010.577,305.135,-150.328,169.300,53.587,160.350
C01484=1010.571,304.887,-150.298,169.294,53.594,160.350
C01485=1010.566,304.639,-150.267,169.286,53.600,160.350
C01486=1010.560,304.391,-150.237,169.281,53.606,160.350
C01487=1010.555,304.142,-150.205,169.274,53.613,160.351
C01488=1010.548,303.895,-150.174,169.267,53.620,160.350
C01489=1010.543,303.647,-150.143,169.261,53.626,160.351
C01490=1010.538,303.399,-150.113,169.254,53.632,160.351
C01491=1010.532,303.151,-150.082,169.247,53.639,160.351
C01492=1010.527,302.903,-150.052,169.242,53.646,160.351
C01493=1010.522,302.655,-150.021,169.234,53.652,160.351
C01494=1010.516,302.407,-149.990,169.228,53.659,160.351
C01495=1010.511,302.159,-149.960,169.221,53.666,160.351
C01496=1010.505,301.910,-149.928,169.215,53.673,160.352
C01497=1010.499,301.663,-149.898,169.208,53.679,160.352
C01498=1010.494,301.415,-149.867,169.201,53.686,160.352
C01499=1010.488,301.167,-149.837,169.196,53.692,160.352
C01500=1010.483,300.919,-149.806,169.189,53.699,160.352
C01501=1010.477,300.671,-149.775,169.182,53.705,160.352
C01502=1010.472,300.423,-149.744,169.176,53.712,160.352
C01503=1010.466,300.175,-149.714,169.169,53.719,160.352
C01504=1010.461,299.927,-149.683,169.163,53.726,160.353
C01505=1010.456,299.679,-149.653,169.157,53.733,160.353
C01506=1010.450,299.431,-149.622,169.150,53.739,160.353
C01507=1010.445,299.184,-149.592,169.143,53.746,160.353
C01508=1010.441,298.935,-149.562,169.137,53.752,160.353
C01509=1010.435,298.687,-149.531,169.131,53.759,160.353
C01510=1010.430,298.439,-149.500,169.124,53.766,160.354
C01511=1010.424,298.191,-149.470,169.118,53.773,160.354
C01512=1010.419,297.942,-149.440,169.112,53.780,160.354
C01513=1010.413,297.694,-149.409,169.106,53.786,160.354
C01514=1010.408,297.446,-149.378,169.099,53.793,160.354
C01515=1010.402,297.199,-149.348,169.093,53.800,160.355
C01516=1010.398,296.950,-149.318,169.086,53.806,160.355
C01517=1010.392,296.703,-149.288,169.080,53.813,160.355
C01518=1010.387,296.455,-149.257,169.073,53.820,160.355
C01519=1010.382,296.206,-149.227,169.067,53.827,160.355
C01520=1010.377,295.958,-149.196,169.061,53.834,160.355
C01521=1010.371,295.711,-149.166,169.054,53.841,160.355
C01522=1010.367,295.462,-149.136,169.049,53.848,160.356
C01523=1010.361,295.214,-149.106,169.042,53.855,160.356
C01524=1010.356,294.965,-149.076,169.035,53.862,160.356
C01525=1010.351,294.718,-149.046,169.030,53.868,160.357
C01526=1010.346,294.470,-149.015,169.023,53.875,160.357
C01527=1010.340,294.222,-148.985,169.016,53.882,160.357
C01528=1010.335,293.973,-148.955,169.011,53.889,160.357
C01529=1010.330,293.679,-148.919,169.003,53.897,160.357
C01530=1010.324,293.384,-148.883,168.995,53.905,160.357
C01531=1010.317,293.089,-148.847,168.988,53.913,160.358
C01532=1010.312,292.794,-148.811,168.981,53.922,160.358
C01533=1010.305,292.479,-148.773,168.973,53.931,160.358
C01534=1010.299,292.164,-148.734,168.965,53.940,160.359
C01535=1010.292,291.849,-148.697,168.957,53.948,160.359
C01536=1010.286,291.535,-148.659,168.949,53.957,160.359
C01537=1010.048,292.611,-149.154,168.950,53.989,160.367
C01538=1010.050,292.713,-149.166,168.953,53.986,160.367
C01539=1010.058,293.112,-149.215,168.964,53.975,160.367
C01540=1010.064,293.410,-149.251,168.971,53.967,160.366
C01541=1010.070,293.707,-149.287,168.978,53.959,160.366
C01542=1010.077,294.004,-149.323,168.986,53.950,160.366
C01543=1010.082,294.252,-149.354,168.991,53.943,160.365
C01544=1010.087,294.500,-149.383,168.998,53.936,160.365
C01545=1010.092,294.748,-149.414,169.005,53.929,160.365
C01546=1010.097,294.997,-149.443,169.010,53.923,160.365
C01547=1010.102,295.244,-149.474,169.017,53.916,160.365
C01548=1010.107,295.492,-149.504,169.024,53.909,160.365
C01549=1010.112,295.741,-149.535,169.030,53.902,160.364
C01550=1010.118,295.989,-149.564,169.036,53.895,160.364
C01551=1010.122,296.236,-149.595,169.043,53.888,160.364
C01552=1010.128,296.485,-149.624,169.049,53.882,160.364
C01553=1010.133,296.733,-149.655,169.055,53.875,160.364
C01554=1010.139,296.981,-149.686,169.062,53.868,160.363
C01555=1010.143,297.229,-149.716,169.068,53.861,160.363
C01556=1010.149,297.477,-149.746,169.074,53.854,160.363
C01557=1010.154,297.725,-149.777,169.081,53.847,160.363
C01558=1010.159,297.974,-149.807,169.087,53.841,160.363
C01559=1010.164,298.221,-149.837,169.093,53.834,160.362
C01560=1010.169,298.470,-149.868,169.101,53.827,160.363
C01561=1010.175,298.718,-149.898,169.106,53.821,160.362
C01562=1010.179,298.965,-149.929,169.113,53.814,160.362
C01563=1010.185,299.213,-149.959,169.120,53.807,160.362
C01564=1010.190,299.461,-149.990,169.125,53.800,160.362
C01565=1010.196,299.709,-150.020,169.132,53.793,160.362
C01566=1010.201,299.958,-150.051,169.139,53.786,160.361
C01567=1010.207,300.206,-150.081,169.145,53.781,160.361
C01568=1010.212,300.454,-150.112,169.152,53.774,160.361
C01569=1010.218,300.702,-150.142,169.158,53.767,160.361
C01570=1010.223,300.950,-150.173,169.165,53.760,160.361
C01571=1010.229,301.198,-150.203,169.171,53.754,160.361
C01572=1010.234,301.446,-150.234,169.178,53.747,160.361
C01573=1010.239,301.694,-150.265,169.185,53.740,160.361
C01574=1010.245,301.942,-150.296,169.190,53.733,160.360
C01575=1010.250,302.190,-150.326,169.197,53.727,160.360
C01576=1010.255,302.438,-150.357,169.204,53.720,160.360
C01577=1010.261,302.686,-150.387,169.210,53.714,160.360
C01578=1010.266,302.934,-150.418,169.217,53.707,160.360
C01579=1010.272,303.182,-150.449,169.224,53.700,160.360
C01580=1010.277,303.430,-150.480,169.230,53.693,160.360
C01581=1010.283,303.677,-150.510,169.237,53.688,160.360
C01582=1010.288,303.926,-150.541,169.243,53.681,160.360
C01583=1010.295,304.174,-150.572,169.250,53.674,160.359
C01584=1010.300,304.422,-150.603,169.256,53.668,160.359
C01585=1010.305,304.670,-150.633,169.263,53.661,160.359
C01586=1010.310,304.918,-150.664,169.270,53.655,160.359
C01587=1010.317,305.165,-150.695,169.276,53.648,160.359
C01588=1010.322,305.414,-150.726,169.283,53.642,160.359
C01589=1010.328,305.662,-150.757,169.290,53.635,160.359
C01590=1010.333,305.910,-150.788,169.297,53.629,160.359
C01591=1010.339,306.157,-150.819,169.303,53.622,160.359
C01592=1010.344,306.406,-150.850,169.310,53.616,160.359
C01593=1010.350,306.653,-150.880,169.316,53.609,160.359
C01594=1010.356,306.902,-150.911,169.324,53.603,160.359
C01595=1010.362,307.149,-150.942,169.329,53.596,160.358
C01596=1010.367,307.398,-150.973,169.337,53.590,160.358
C01597=1010.373,307.645,-151.004,169.343,53.583,160.358
C01598=1010.379,307.894,-151.036,169.349,53.577,160.358
C01599=1010.386,308.209,-151.075,169.359,53.568,160.358
C01600=1010.393,308.524,-151.114,169.367,53.561,160.358
C01601=1010.401,308.840,-151.154,169.376,53.552,160.358
C01602=1010.407,309.155,-151.195,169.384,53.544,160.358
C01603=1010.413,309.402,-151.226,169.391,53.539,160.358
C01604=1010.418,309.650,-151.258,169.397,53.532,160.358
C01605=1010.424,309.898,-151.290,169.404,53.525,160.358
C01606=1010.429,310.146,-151.322,169.411,53.520,160.358
C01607=1010.434,310.393,-151.354,169.418,53.513,160.358
C01608=1010.440,310.642,-151.386,169.425,53.507,160.358
C01609=1010.445,310.889,-151.418,169.431,53.501,160.358
C01610=1010.451,311.138,-151.449,169.438,53.494,160.358
C01611=1010.456,311.386,-151.481,169.445,53.488,160.358
C01612=1010.461,311.633,-151.513,169.451,53.482,160.358
C01613=1010.467,311.882,-151.545,169.458,53.476,160.358
C01614=1010.472,312.129,-151.576,169.466,53.470,160.358
C01615=1010.478,312.377,-151.609,169.472,53.464,160.358
C01616=1010.484,312.624,-151.641,169.479,53.458,160.358
C01617=1010.489,312.872,-151.673,169.486,53.451,160.358
C01618=1010.495,313.120,-151.705,169.492,53.446,160.358
C01619=1010.500,313.368,-151.737,169.500,53.439,160.358
C01620=1010.506,313.616,-151.769,169.507,53.433,160.358
C01621=1010.511,313.863,-151.801,169.514,53.427,160.358
C01622=1010.517,314.112,-151.833,169.520,53.421,160.358
C01623=1010.523,314.359,-151.864,169.527,53.415,160.358
C01624=1010.528,314.607,-151.898,169.534,53.409,160.358
C01625=1010.534,314.855,-151.930,169.541,53.403,160.358
C01626=1010.540,315.103,-151.961,169.548,53.397,160.358
C01627=1010.546,315.351,-151.993,169.555,53.390,160.358
C01628=1010.551,315.598,-152.026,169.562,53.384,160.358
C01629=1010.557,315.846,-152.058,169.568,53.378,160.358
C01630=1010.563,316.095,-152.090,169.576,53.372,160.358
C01631=1010.568,316.342,-152.122,169.583,53.366,160.358
C01632=1010.574,316.590,-152.155,169.589,53.361,160.359
C01633=1010.580,316.838,-152.187,169.597,53.354,160.359
C01634=1010.586,317.086,-152.218,169.604,53.348,160.359
C01635=1010.592,317.333,-152.251,169.611,53.342,160.359
C01636=1010.597,317.582,-152.284,169.617,53.336,160.359
C01637=1010.603,317.829,-152.316,169.625,53.331,160.359
C01638=1010.609,318.077,-152.348,169.632,53.324,160.359
C01639=1010.615,318.324,-152.381,169.639,53.318,160.359
C01640=1010.621,318.573,-152.413,169.645,53.312,160.359
C01641=1010.626,318.820,-152.446,169.653,53.307,160.359
C01642=1010.632,319.068,-152.478,169.660,53.301,160.359
C01643=1010.638,319.316,-152.511,169.667,53.294,160.359
C01644=1010.644,319.564,-152.543,169.674,53.289,160.360
C01645=1010.651,319.811,-152.575,169.681,53.283,160.360
C01646=1010.656,320.059,-152.607,169.688,53.277,160.360
C01647=1010.662,320.307,-152.640,169.696,53.271,160.360
C01648=1010.668,320.554,-152.673,169.702,53.266,160.360
C01649=1010.674,320.803,-152.705,169.709,53.259,160.360
C01650=1010.680,321.050,-152.738,169.717,53.254,160.360
C01651=1010.687,321.298,-152.771,169.724,53.248,160.360
C01652=1010.693,321.546,-152.803,169.731,53.242,160.360
C01653=1010.698,321.794,-152.836,169.738,53.236,160.361
C01654=1010.704,322.041,-152.869,169.746,53.231,160.361
C01655=1010.711,322.289,-152.902,169.753,53.225,160.361
C01656=1010.717,322.537,-152.934,169.761,53.219,160.361
C01657=1010.723,322.785,-152.966,169.767,53.213,160.361
C01658=1010.729,323.033,-153.000,169.775,53.208,160.361
C01659=1010.736,323.353,-153.041,169.783,53.200,160.361
C01660=1010.744,323.674,-153.084,169.793,53.193,160.362
C01661=1010.752,323.996,-153.127,169.802,53.185,160.362
C01662=1010.761,324.316,-153.169,169.812,53.178,160.362
C01663=1010.767,324.564,-153.202,169.820,53.172,160.362
C01664=1010.773,324.812,-153.235,169.826,53.166,160.362
C01665=1010.779,325.059,-153.268,169.834,53.161,160.363
C01666=1010.785,325.307,-153.301,169.842,53.155,160.363
C01667=1010.791,325.555,-153.334,169.849,53.149,160.363
C01668=1010.797,325.802,-153.367,169.855,53.144,160.363
C01669=1010.803,326.050,-153.401,169.863,53.138,160.363
C01670=1010.809,326.297,-153.434,169.871,53.133,160.364
C01671=1010.816,326.546,-153.467,169.878,53.127,160.364
C01672=1010.821,326.793,-153.501,169.886,53.121,160.364
C01673=1010.827,327.041,-153.535,169.892,53.116,160.364
C01674=1010.833,327.289,-153.567,169.900,53.111,160.364
C01675=1010.839,327.536,-153.601,169.908,53.105,160.365
C01676=1010.845,327.784,-153.635,169.915,53.099,160.365
C01677=1010.852,328.031,-153.669,169.922,53.094,160.365
C01678=1010.857,328.279,-153.702,169.929,53.089,160.365
C01679=1010.864,328.526,-153.735,169.937,53.083,160.366
C01680=1010.870,328.774,-153.769,169.944,53.077,160.366
C01681=1010.876,329.022,-153.803,169.952,53.072,160.366
C01682=1010.882,329.270,-153.836,169.959,53.067,160.366
C01683=1010.888,329.517,-153.870,169.966,53.061,160.366
C01684=1010.894,329.766,-153.904,169.974,53.056,160.367
C01685=1010.901,330.013,-153.937,169.982,53.050,160.367
C01686=1010.907,330.261,-153.970,169.990,53.045,160.367
C01687=1010.913,330.509,-154.005,169.997,53.040,160.368
C01688=1010.920,330.755,-154.038,170.004,53.035,160.368
C01689=1010.925,331.003,-154.072,170.012,53.029,160.368
C01690=1010.932,331.251,-154.106,170.019,53.024,160.368
C01691=1010.938,331.498,-154.140,170.027,53.018,160.369
C01692=1010.945,331.746,-154.174,170.035,53.013,160.369
C01693=1010.951,331.994,-154.208,170.042,53.007,160.369
C01694=1010.956,332.241,-154.242,170.049,53.003,160.369
C01695=1010.963,332.489,-154.277,170.057,52.997,160.370
C01696=1010.969,332.736,-154.309,170.065,52.992,160.370
C01697=1010.976,332.984,-154.344,170.072,52.986,160.370
C01698=1010.981,333.232,-154.378,170.081,52.981,160.371
C01699=1010.988,333.480,-154.412,170.088,52.976,160.371
C01700=1010.994,333.727,-154.446,170.095,52.971,160.371
C01701=1011.001,333.974,-154.481,170.102,52.965,160.371
C01702=1011.006,334.222,-154.515,170.111,52.960,160.372
C01703=1011.013,334.470,-154.550,170.118,52.955,160.372
C01704=1011.019,334.717,-154.584,170.126,52.950,160.373
C01705=1011.025,334.965,-154.618,170.134,52.944,160.373
C01706=1011.032,335.212,-154.652,170.141,52.939,160.373
C01707=1011.038,335.460,-154.686,170.149,52.934,160.373
C01708=1011.045,335.707,-154.721,170.156,52.929,160.374
C01709=1011.051,335.955,-154.755,170.165,52.924,160.374
C01710=1011.057,336.202,-154.790,170.172,52.919,160.374
C01711=1011.064,336.450,-154.824,170.180,52.914,160.375
C01712=1011.070,336.697,-154.859,170.188,52.908,160.375
C01713=1011.076,336.945,-154.893,170.196,52.904,160.376
C01714=1011.083,337.193,-154.928,170.203,52.898,160.376
C01715=1011.089,337.440,-154.963,170.211,52.894,160.376
C01716=1011.096,337.687,-154.996,170.218,52.888,160.377
C01717=1011.103,337.935,-155.031,170.227,52.883,160.377
C01718=1011.110,338.183,-155.066,170.234,52.878,160.377
C01719=1011.117,338.499,-155.111,170.244,52.872,160.378
C01720=1011.126,338.816,-155.155,170.255,52.866,160.379
C01721=1011.133,339.132,-155.200,170.265,52.859,160.379
C01722=1011.142,339.449,-155.244,170.275,52.853,160.380
C01723=1011.149,339.696,-155.279,170.282,52.847,160.380
C01724=1011.155,339.944,-155.314,170.290,52.843,160.380
C01725=1011.160,340.191,-155.349,170.298,52.838,160.381
C01726=1011.167,340.439,-155.384,170.306,52.833,160.381
C01727=1011.174,340.686,-155.419,170.314,52.828,160.382
C01728=1011.180,340.934,-155.454,170.322,52.823,160.382
C01729=1011.187,341.181,-155.489,170.330,52.818,160.382
C01730=1011.194,341.429,-155.524,170.338,52.813,160.383
C01731=1011.200,341.676,-155.560,170.346,52.808,160.383
C01732=1011.207,341.924,-155.595,170.355,52.803,160.384
C01733=1011.214,342.171,-155.630,170.363,52.799,160.384
C01734=1011.220,342.419,-155.665,170.371,52.794,160.385
C01735=1011.227,342.666,-155.700,170.379,52.789,160.385
C01736=1011.233,342.914,-155.736,170.387,52.784,160.386
C01737=1011.240,343.161,-155.771,170.394,52.780,160.386
C01738=1011.247,343.408,-155.806,170.402,52.775,160.386
C01739=1011.253,343.656,-155.842,170.410,52.770,160.387
C01740=1011.259,343.903,-155.877,170.418,52.765,160.387
C01741=1011.266,344.151,-155.912,170.426,52.760,160.388
C01742=1011.273,344.398,-155.948,170.435,52.756,160.388
C01743=1011.280,344.645,-155.983,170.443,52.751,160.389
C01744=1011.286,344.893,-156.019,170.451,52.746,160.389
C01745=1011.293,345.140,-156.054,170.459,52.741,160.390
C01746=1011.300,345.387,-156.089,170.467,52.737,160.390
C01747=1011.306,345.635,-156.125,170.476,52.732,160.391
C01748=1011.313,345.882,-156.161,170.484,52.727,160.391
C01749=1011.320,346.130,-156.197,170.492,52.723,160.392
C01750=1011.327,346.377,-156.232,170.500,52.718,160.392
C01751=1011.333,346.624,-156.268,170.508,52.714,160.393
C01752=1011.340,346.872,-156.303,170.517,52.709,160.393
C01753=1011.347,347.119,-156.340,170.525,52.704,160.394
C01754=1011.354,347.367,-156.375,170.533,52.700,160.395
C01755=1011.360,347.614,-156.412,170.541,52.695,160.395
C01756=1011.367,347.861,-156.447,170.549,52.690,160.396
C01757=1011.374,348.109,-156.484,170.558,52.686,160.396
C01758=1011.381,348.356,-156.519,170.566,52.681,160.397
C01759=1011.387,348.603,-156.555,170.575,52.677,160.397
C01760=1011.394,348.850,-156.591,170.583,52.672,160.398
C01761=1011.401,349.098,-156.628,170.591,52.668,160.399
C01762=1011.408,349.345,-156.663,170.599,52.663,160.399
C01763=1011.414,349.592,-156.699,170.608,52.659,160.400
C01764=1011.422,349.840,-156.736,170.617,52.654,160.400
C01765=1011.428,350.087,-156.772,170.626,52.650,160.401
C01766=1011.436,350.334,-156.808,170.634,52.645,160.401
C01767=1011.442,350.582,-156.844,170.642,52.641,160.402
C01768=1011.449,350.829,-156.880,170.651,52.637,160.403
C01769=1011.456,351.076,-156.917,170.659,52.632,160.403
C01770=1011.463,351.323,-156.953,170.667,52.628,160.404
C01771=1011.470,351.571,-156.989,170.676,52.624,160.405
C01772=1011.477,351.818,-157.025,170.684,52.619,160.405
C01773=1011.484,352.065,-157.062,170.693,52.615,160.406
C01774=1011.491,352.312,-157.098,170.701,52.610,160.406
C01775=1011.498,352.560,-157.135,170.709,52.606,160.407
C01776=1011.505,352.807,-157.171,170.719,52.601,160.408
C01777=1011.512,353.054,-157.207,170.727,52.597,160.408
